// ---- FunctionBlocks/Sorter/Functions/FB_SorterLog.TcPOU
FUNCTION_BLOCK FB_SorterLog
VAR_IN_OUT
END_VAR
VAR_INPUT
	SorterToLog			:	ST_Sorter;
	SorterLogEnable		:	UDINT;
	ToInduct			:	ST_ItemTemporary;
END_VAR
VAR_OUTPUT
	TempItem			:	ST_ItemTemporary;
END_VAR
VAR
	rInductPE			:	R_TRIG;
	fInductPE			:	F_TRIG;
	rDischargePE		:	R_TRIG;
	fDischargePE		:	F_TRIG;
	sMessage			:	STRING;
	BlankItem			: 	ST_Item := (ID := ''
										, UniqueID := 0
										, Destination := 0
										, Status := E_StatusCode.No_Status
										, ExtStatus := E_StatusCode.No_Status
										, DeviceID := ''
										, MessageType := E_MessageIds.NoMessage_00);
END_VAR

// Capture rising and falling edge Triggers of the configured Sorter PE (Induct/Discharge)
rInductPE(CLK:= SorterToLog.InductPE, Q =>);
fInductPE(CLK:= SorterToLog.InductPE, Q =>);
rDischargePE(CLK:= SorterToLog.DischargePE, Q =>);
fDischargePE(CLK:= SorterToLog.DischargePE, Q =>);

// On the rising/falling edge of the Induct PE
IF rInductPE.Q OR fInductPE.Q THEN
	IF SorterLogEnable.SORTER_DISCHARGE_PE THEN
		// Write to the Error List
		ADSLOGSTR( msgCtrlMask := ADSLOG_MSGTYPE_HINT OR ADSLOG_MSGTYPE_LOG
			, msgFmtStr := CONCAT(sortertolog.Config.Name,' Induct PE Blocked : %s')
			, strArg := BOOL_TO_STRING(SorterToLog.InductPE)); 
	END_IF
END_IF

// Prepare a dummy record for items that arrive before BCR data is received
// On the rising edge of the Induct PE
IF rInductPE.Q THEN
	// Test for a UniqueID, which indicates that a Barcode has been received
	IF ToInduct.Item.UniqueID = 0 THEN
		// Capture and create relevant info
		TempItem.Counts := SorterToLog.EncoderCounts;
		TempItem.Item.UniqueID :=  UDINT_TO_DINT(SorterToLog.EncoderCounts);
		TempItem.Item.ID :=  CONCAT('T-', UDINT_TO_STRING(SorterToLog.EncoderCounts));
		TempItem.Item.Destination := SorterToLog.Config.DefaultDestination;
		TempItem.Item.DestinationIdx := SorterToLog.Config.DefaultDestIdx;
		TempItem.Item.Status := E_StatusCode.UnidentifiedItem;
		IF SorterLogEnable.SORTER_TEMPID THEN
			ADSLOGSTR( msgCtrlMask := ADSLOG_MSGTYPE_HINT OR ADSLOG_MSGTYPE_LOG
				, msgFmtStr := CONCAT(sortertolog.Config.Name,' Temp ID Assigned : %s')
				, strArg := TempItem.Item.ID);
		END_IF
	END_IF	
END_IF

// Clear the dummy record when the PE clears
// Items can only be inducted when the BCR info is received before or while the induct PE is blocked
IF fInductPE.Q THEN
	// Clear the record
	TempItem.Counts := 0;
	TempItem.Item :=  BlankItem;
END_IF

// On the rising/falling edge of the Discharge PE
IF rDischargePE.Q OR fDischargePE.Q THEN
	IF SorterLogEnable.SORTER_DISCHARGE_PE THEN
		// Write to the Error List
		ADSLOGSTR( msgCtrlMask := ADSLOG_MSGTYPE_HINT OR ADSLOG_MSGTYPE_LOG
			, msgFmtStr := CONCAT(sortertolog.Config.Name,' Discharge PE Blocked : %s')
			, strArg := BOOL_TO_STRING(SorterToLog.DischargePE)); 
	END_IF
END_IF

END_FUNCTION_BLOCK

// ---- FunctionBlocks/Divert/Functions/FB_DivertLog.TcPOU
FUNCTION_BLOCK FB_DivertLog
VAR_IN_OUT
	DivertArray	: ARRAY[*] OF ST_Divert;
END_VAR
VAR_INPUT
	DivertLogEnable		:	UDINT;
	EncoderCounts		:	UDINT;
END_VAR
VAR_OUTPUT
END_VAR
VAR
	DivertCountMax			: DINT;
	DivertCountMin			: DINT;
	DivertIndex				: DINT;
	r_DivertExtend			: ARRAY [1..16] OF R_TRIG;
	f_DivertExtend			: ARRAY [1..16] OF F_TRIG;
	r_ConfirmPE				: ARRAY [1..16] OF R_TRIG;
	f_ConfirmPE				: ARRAY [1..16] OF F_TRIG;
	sMessage				: STRING;
END_VAR

// Get the Max and Min counts
DivertCountMin := LOWER_BOUND(DivertArray,1);
DivertCountMax := UPPER_BOUND(DivertArray,1);

FOR DivertIndex := DivertCountMin TO DivertCountMax DO
	// Divert at DivertIndex
	r_DivertExtend[DivertIndex](CLK := DivertArray[DivertIndex].Output1);
	f_DivertExtend[DivertIndex](CLK := DivertArray[DivertIndex].Output1);
	
	IF r_DivertExtend[DivertIndex].Q THEN
		// Mask the divert index to see if it should be logged
		IF ((DivertLogEnable AND LREAL_TO_UDINT(EXPT(2,DivertIndex))) > 0) THEN
			sMessage := DINT_TO_STRING(DivertIndex);
			sMessage := CONCAT(sMessage,' : ');
			sMessage := CONCAT(sMessage, UDINT_TO_STRING(EncoderCounts));
			ADSLOGSTR( msgCtrlMask := ADSLOG_MSGTYPE_HINT OR ADSLOG_MSGTYPE_LOG
				, msgFmtStr := CONCAT(DivertArray[DivertIndex].Config.ID, ' Extend Divert %s')
				, strArg := sMessage); 
		END_IF;
	END_IF
	IF f_DivertExtend[DivertIndex].Q THEN
		// Mask the divert index to see if it should be logged
		IF ((DivertLogEnable AND LREAL_TO_UDINT(EXPT(2,DivertIndex))) > 0) THEN
			sMessage := DINT_TO_STRING(DivertIndex);
			sMessage := CONCAT(sMessage,' : ');
			sMessage := CONCAT(sMEssage, UDINT_TO_STRING(EncoderCounts));
			ADSLOGSTR( msgCtrlMask := ADSLOG_MSGTYPE_HINT OR ADSLOG_MSGTYPE_LOG
				, msgFmtStr := CONCAT(DivertArray[DivertIndex].Config.ID, ' Retract Divert %s')
				, strArg := sMessage); 
		END_IF;
	END_IF
	
	// Confirm at DivertIndex
	r_ConfirmPE[DivertIndex](CLK := DivertArray[DivertIndex].ConfirmPE);
	f_ConfirmPE[DivertIndex](CLK := DivertArray[DivertIndex].ConfirmPE);
	
	IF r_ConfirmPE[DivertIndex].Q THEN
		// Mask the convirm index to see if it should be logged
		IF ((DivertLogEnable AND LREAL_TO_UDINT(EXPT(2,(DivertIndex+15)))) > 0) THEN
			sMessage := DINT_TO_STRING(DivertIndex);
			sMessage := CONCAT(sMessage,' Blocked: ');
			sMessage := CONCAT(sMEssage, UDINT_TO_STRING(EncoderCounts));
			ADSLOGSTR( msgCtrlMask := ADSLOG_MSGTYPE_HINT OR ADSLOG_MSGTYPE_LOG
				, msgFmtStr := CONCAT(DivertArray[DivertIndex].Config.ID, ' Configm PE %s')
				, strArg := sMessage); 
		END_IF;
	END_IF
	IF f_ConfirmPE[DivertIndex].Q THEN
		// Mask the convirm index to see if it should be logged
		IF ((DivertLogEnable AND LREAL_TO_UDINT(EXPT(2,(DivertIndex+15)))) > 0) THEN
			sMessage := DINT_TO_STRING(DivertIndex);
			sMessage := CONCAT(sMessage,' Cleared: ');
			sMessage := CONCAT(sMEssage, UDINT_TO_STRING(EncoderCounts));
			ADSLOGSTR( msgCtrlMask := ADSLOG_MSGTYPE_HINT OR ADSLOG_MSGTYPE_LOG
				, msgFmtStr := CONCAT(DivertArray[DivertIndex].Config.ID, ' Configm PE %s')
				, strArg := sMessage); 
		END_IF;
	END_IF
END_FOR

END_FUNCTION_BLOCK

// ---- POUs/ProcessBuffers_P2140.TcPOU
PROGRAM ProcessBuffers_P2140
VAR_IN_OUT
	st_NextToInduct					: ST_ItemTemporary;
	st_UpdateItem					: ST_ItemTemporary;
	st_TempInductItem				: ST_ItemTemporary;
	{attribute 'OPC.UA.DA' := '0'}
	st_Sorter						: ST_Sorter;
	{attribute 'OPC.UA.DA' := '0'}
	aDiverts						: ARRAY[Sorter.DIVERTMIN_P2140..Sorter.NUMBEROFDIVERTS_P2140] OF ST_DIVERT;
	aItems 							: ARRAY[Sorter.SORTERENCODERMIN_P2140..Sorter.SORTERENCODERMAX_P2140] OF ST_Item;
END_VAR

VAR_INPUT
	DestinationOverride				: DINT;	// Pass in Divert to sent item to regardless of the direction received
	DivertToCommission				: DINT;
	ItemsArrayMax 					: UDINT;
	ItemsArrayMin 					: UDINT;
END_VAR

VAR_OUTPUT
	DefaultDestIdx					: DINT;
	RecircDestIdx					: DINT;
END_VAR

VAR
	fb_ArrivalBuffer				: FB_ItemBuffer;
	st_ArrivalItem 					: ST_Item;		// Arrival Item (Bar code read) from System PLC (BarCodeReaders.pou)

	// Item to replace in the sorter buffer
	st_ReplaceItem					: st_Item;

	fb_TransportBuffer				: FB_ItemBuffer;

	fb_UpdateBuffer 				: FB_ItemBuffer;

	st_ToUpdate						: ST_ItemTemporary;	// Item to Update on the Sorter, or waiting to be added to the sorter

	ItemsArraySize			: UDINT;

	TransportItemInSorter	: ST_Item;	// Temporary Processing Item
	TransportItemFound		: ST_Item;	// Item to Update Found
	TransportSorterIndex	: UDINT;

	ExitSorterIndex			: UDINT;
	ExitItemInSorter		: ST_Item;
	ExitItemFound			: ST_ItemTemporary;
	ExitInDivert			: BOOL;
	ExitDiverting			: BOOL;
	ExitSuccess				: BOOL;
	ExitDetected			: BOOL;
	ExitComplete			: BOOL;

	UpdateIndexCounter		: DINT;

	bTest : BOOL;
	sMessage	:	STRING;
	
	st_DisplayItem		:st_Item;
	LogSorterDump		:BOOL := FALSE;

	fb_FindDestination		: FB_FindDestination;
	fb_DefaultDestination	: FB_FindDestination;
	fb_RecircDestination	: FB_FindDestination;
	// Created to allow the aDiverts to be used in the FB_FindDestination Function Block
	{attribute 'OPC.UA.DA' := '0'}
	aTempDiverts			: ARRAY[Sorter.DIVERTMIN_P2140..Sorter.NUMBEROFDIVERTS_P2140] OF ST_DIVERT;
	
	nItemBufferLogEnable	:	UDINT;
	nSorterLogEnable		:	UDINT;
	nDivertLogEnable		:	UDINT;
	nSortBufferLogEnable	:	UDINT;
END_VAR

nItemBufferLogEnable := GVL_Logging.nItemBufferLogEnable OR GVL_Logging.nItemBufferLogEnableP2140;
nSorterLogEnable := GVL_Logging.nSorterLogEnable OR GVL_Logging.nSorterLogEnableP2140;
nDivertLogEnable := GVL_Logging.nDivertLogEnable OR GVL_Logging.nDivertLogEnableP2140;
nSortBufferLogEnable := GVL_Logging.nSortBufferLogEnable OR GVL_Logging.nSortBufferLogEnableP2140;

aTempDiverts := aDiverts;
// Initialize the Transport and Update buffers
// Set Master for FB's that control the buffer
fb_ArrivalBuffer.Master := FALSE;
fb_TransportBuffer.Master := FALSE;
fb_UpdateBuffer.Master := FALSE;

// Turn ON/OFF Logging of all activity in/out
fb_ArrivalBuffer.LogEntries := nItemBufferLogEnable.ARRIVALS;
fb_TransportBuffer.LogEntries := nItemBufferLogEnable.TRANSPORT;
fb_UpdateBuffer.LogEntries := nItemBufferLogEnable.UPDATE;

// Provide names for the buffers
fb_ArrivalBuffer.Name := CONCAT(st_Sorter.Config.Name, ' SRT ARRIVAL');
fb_TransportBuffer.Name := CONCAT(st_Sorter.Config.Name, ' SRT TRANSPORT');
fb_UpdateBuffer.Name := CONCAT(st_Sorter.Config.Name, ' SRT UPDATE');

// Initialize the FB_ItemExtBuffer Instances
fb_ArrivalBuffer(st_BufferData := st_SorterArrivalBuffer_P2140
						, st_BufferFdbkIn := st_ArrivalFdbkOut_P2140
						, st_BufferFdbkOut => st_ArrivalFdbkIn_P2140);
fb_TransportBuffer(st_BufferData := st_SorterTransportBuffer_P2140
						, st_BufferFdbkIn := st_TransportFdbkOut_P2140
						, st_BufferFdbkOut => st_TransportFdbkIn_P2140);
fb_UpdateBuffer(st_BufferData := st_SorterUpdateBuffer
						, st_BufferFdbkIn := st_UpdateFdbkOut
						, st_BufferFdbkOut => st_UpdateFdbkIn);

IF GVL_IO.INIT THEN
	fb_ArrivalBuffer.Clear();
	fb_TransportBuffer.Clear();
	fb_UpdateBuffer.Clear();
END_IF
						
(*
	Set the Upper/Lower bound of relevant arrays for looping purposes
	ItemsArrayMax/Min for the sorter array slot count
*)
// Size is Max - Min + 1 to capture both extremes
ItemsArraySize := ItemsArrayMax - ItemsArrayMin + 1;

(*
 	Check for a value disagreement in the Arrival Buffer In and Out pointers to
  	determine if there is an update for an item.
	When an Item arrives, the System PLC adds it to the shared buffer and increments
	the InPointer
*)
IF st_SorterArrivalBuffer_P2140.nInPointer <> fb_ArrivalBuffer.OutPointer THEN
	fb_ArrivalBuffer.RemoveItem(st_ItemToReturn => st_ArrivalItem);
END_IF

// Input Item read at bar code reader from System PLC to sorter
IF st_ArrivalItem.ID <> '' THEN
	IF nSortBufferLogEnable.BUFFER_ARRIVAL THEN
		sMessage := CONCAT('Item: ', st_ArrivalItem.ID);
		sMessage := CONCAT(sMessage,' Pulses: ');
		sMessage := CONCAT(sMessage, UDINT_TO_STRING(st_Sorter.EncoderCounts));
		// Write to the Error List
		ADSLOGSTR( msgCtrlMask := ADSLOG_MSGTYPE_HINT OR ADSLOG_MSGTYPE_LOG
			, msgFmtStr := CONCAT(st_Sorter.Config.Name, ' Arrival Processed: %s')
			, strArg := sMessage);
	END_IF
	// Indicate that this item did not get added to the sorter and add to the exit buffer
	//  Both as a TransportUpdate and TransportComplete message type 
	IF st_NextToInduct.Item.ID <> '' THEN
		IF nSortBufferLogEnable.BUFFER_MISSINDUCT THEN
			sMessage := CONCAT('Item: ', st_NextToInduct.Item.ID);
			// Write to the Error List
			ADSLOGSTR( msgCtrlMask := ADSLOG_MSGTYPE_HINT OR ADSLOG_MSGTYPE_LOG
				, msgFmtStr := CONCAT(st_Sorter.Config.Name, ' Item Removed - Not Inducted: %s')
				, strArg := sMessage);
		END_IF
		// Transport Response
		st_NextToInduct.Item.Status := E_StatusCode.Assign_NotInducted;
		st_NextToInduct.Item.DeviceID := st_Sorter.Config.EquipID;
		st_NextToInduct.Item.MessageType := E_MessageIds.TransportResponse_25;
		fb_UpdateBuffer.AddItem(st_ItemToAdd := st_NextToInduct.Item);

		// Transport Complete
		st_NextToInduct.Item.Status := E_StatusCode.Divert_NotInducted;
		st_NextToInduct.Item.MessageType := E_MessageIds.TransportComplete_26;
		fb_UpdateBuffer.AddItem(st_ItemToAdd := st_NextToInduct.Item);
	END_IF
	// Copy Last BCR item to Item to Induct
	st_NextToInduct.Item :=  st_ArrivalItem;
	// Add the Sorter EquipID to the NextToInduct
	st_NextToInduct.Item.DeviceID := st_Sorter.Config.EquipID;
	// Set the Default Destination
	IF DestinationOverride = 0 THEN
		st_NextToInduct.Item.Destination := st_Sorter.Config.DefaultDestination;
		st_NextToInduct.Item.DestinationIdx := st_Sorter.Config.DefaultDestIdx;
	ELSE
		st_NextToInduct.Item.Destination := DestinationOverride;
		IF nSorterLogEnable.SORTER_DESTINATION_LU THEN
			sMessage := CONCAT('Destination: ', DINT_TO_STRING(st_NextToInduct.Item.Destination));
			// Write to the Error List
			ADSLOGSTR( msgCtrlMask := ADSLOG_MSGTYPE_HINT OR ADSLOG_MSGTYPE_LOG
				, msgFmtStr := CONCAT(st_sorter.Config.Name, ' Buffer Destination OR Lookup %s')
				, strArg := sMessage);
		END_IF
		fb_FindDestination(RoundRobin := st_Sorter.RoundRobin
						, SorterLogEnable := nSorterLogEnable
						, aDiverts := aTempDiverts
						, DestinationID := st_NextToInduct.Item.Destination
						, DestinationIndex => st_NextToInduct.Item.DestinationIdx);
		
	END_IF
	// Capture an encoder value that when the encoder count exceeds this value, NextToInduct item will be cleared
	st_NextToInduct.Counts := st_Sorter.EncoderCounts;
	// Clear the Last recieved item
	st_ArrivalItem := BlankItem;
	// Prepare to replace the Temporarily assigned item with this item
	IF st_TempInductItem.Item.ID <> '' THEN
		// Capture the Counts and Length from the temporary item
		st_NextToInduct.Counts := st_TempInductItem.Counts;
		st_NextToInduct.Item.Length := st_TempInductItem.Item.Length;
		//Identify the Item to replace in the sorter array
		st_ReplaceItem := st_TempInductItem.Item;
		st_TempInductItem.Counts := 0;
		st_TempInductItem.Item := BlankItem;
		IF nSortBufferLogEnable.BUFFER_TEMPINDUCT THEN
			ADSLOGSTR( msgCtrlMask := ADSLOG_MSGTYPE_HINT OR ADSLOG_MSGTYPE_LOG
				, msgFmtStr := CONCAT(st_Sorter.Config.Name, ' Temp ID Replaced : %s')
				, strArg := st_ReplaceItem.ID); 
		END_IF
	END_IF
END_IF

(*
 	Check for a value disagreement in the SorterTransportBuffer In and Out pointers to
  	determine if there is an update for an item.
	When an update arrived, the System PLC adds it to the shared buffer and increments
	the InPointer
*)
IF st_SorterTransportBuffer_P2140.nInPointer <> fb_TransportBuffer.OutPointer THEN
	fb_TransportBuffer.RemoveItem(st_ItemToReturn => st_ToUpdate.Item);
	// Override any received destination if there is an Override
	IF DestinationOverride <> 0 THEN
		st_ToUpdate.Item.Destination := DestinationOverride;
	END_IF
	// Lookup the index for the chosen destination
	IF nSorterLogEnable.SORTER_DESTINATION_LU THEN
		sMessage := CONCAT('Destination: ', DINT_TO_STRING(st_ToUpdate.Item.Destination));
		// Write to the Error List
		ADSLOGSTR( msgCtrlMask := ADSLOG_MSGTYPE_HINT OR ADSLOG_MSGTYPE_LOG
			, msgFmtStr := CONCAT(st_sorter.Config.Name, ' Buffer Update Lookup %s')
			, strArg := sMessage);
	END_IF
	fb_FindDestination(RoundRobin := st_Sorter.RoundRobin
					, SorterLogEnable := nSorterLogEnable
					, aDiverts := aTempDiverts
					, DestinationID := st_ToUpdate.Item.Destination
					, DestinationIndex => st_ToUpdate.Item.DestinationIdx);
	IF nSortBufferLogEnable.BUFFER_DESTINDEX THEN
		sMessage := CONCAT('Item: ', st_ToUpdate.Item.ID);
		sMessage := CONCAT(sMessage,' Destination: ');
		sMessage := CONCAT(sMessage, DINT_TO_STRING(st_ToUpdate.Item.Destination));
		sMessage := CONCAT(sMessage,' Index: ');
		sMessage := CONCAT(sMessage, DINT_TO_STRING(st_ToUpdate.Item.DestinationIdx));
		// Write to the Error List
		ADSLOGSTR( msgCtrlMask := ADSLOG_MSGTYPE_HINT OR ADSLOG_MSGTYPE_LOG
			, msgFmtStr := CONCAT(st_Sorter.Config.Name, ' Divert Index of Destination: %s')
			, strArg := sMessage);
	END_IF
END_IF

// Get the Default Destination Index
fb_DefaultDestination(RoundRobin := st_Sorter.RoundRobin
				, NoAssignment := TRUE
				, aDiverts := aTempDiverts
				, DestinationID := st_Sorter.Config.DefaultDestination
				, DestinationIndex => DefaultDestIdx);

// Get the Recirculation Destination Index
fb_RecircDestination(RoundRobin := st_Sorter.RoundRobin
				, NoAssignment := TRUE
				, aDiverts := aTempDiverts
				, DestinationID := st_Sorter.Config.RecircDestination
				, DestinationIndex => RecircDestIdx);

// Test the Item to Update against the Item to Induct and update if they match:
//	Update the NextItemToInduct with the updated data, then clear the Item to Update
IF st_ToUpdate.Item.ID <> '' THEN
	IF st_ToUpdate.Item.ID = st_NextToInduct.Item.ID THEN
		// Indicate that the transport command was received and a response was sent
		st_NextToInduct.Item.MessageType := E_MessageIds.TransportResponse_25;
		// Test the assigned lane for availability
		IF (aDiverts[st_ToUpdate.Item.DestinationIdx].Full
		   OR aDiverts[st_ToUpdate.Item.DestinationIdx].Faulted)
		   AND DestinationOverride = 0
		   THEN
			// Prepare a message to indicate that the item cannot be assigned
			st_ToUpdate.Item.Status := E_StatusCode.Assign_Full;
			st_ToUpdate.Item.DeviceID := st_Sorter.Config.EquipID;
			st_ToUpdate.Item.MessageType := E_MessageIds.TransportResponse_25;
			fb_UpdateBuffer.AddItem(st_ItemToAdd := st_ToUpdate.Item);
			st_NextToInduct.Item.ExtStatus := E_StatusCode.Divert_Full;
		ELSE
			st_NextToInduct.Item.DeviceID := st_Sorter.Config.EquipID;
			st_NextToInduct.Item.Status := E_StatusCode.Assign_Accepted;
			// Update the Destination
			st_NextToInduct.Item.Destination := st_ToUpdate.Item.Destination;
			st_NextToInduct.Item.DestinationIdx := st_ToUpdate.Item.DestinationIdx;
			fb_UpdateBuffer.AddItem(st_ItemToAdd := st_NextToInduct.Item);
		END_IF
		// If commissioning, ignore any other direction
		IF DivertToCommission > 0 THEN
			st_NextToInduct.Item.Destination := DivertToCommission;
		END_IF
		// Log the update
		IF nSortBufferLogEnable.BUFFER_INDUCT THEN
			sMessage := CONCAT('Item: ', st_ToUpdate.Item.ID);
			sMessage := CONCAT(sMessage,' Pulses: ');
			sMessage := CONCAT(sMessage, UDINT_TO_STRING(st_Sorter.EncoderCounts));
			sMessage := CONCAT(sMessage,' Status: ');
			sMessage := CONCAT(sMessage, UDINT_TO_STRING(st_ToUpdate.Item.Status));
			sMessage := CONCAT(sMessage,' Ext Status: ');
			sMessage := CONCAT(sMessage, UDINT_TO_STRING(st_ToUpdate.Item.ExtStatus));
			// Write to the Error List
			ADSLOGSTR( msgCtrlMask := ADSLOG_MSGTYPE_HINT OR ADSLOG_MSGTYPE_LOG
				, msgFmtStr := CONCAT(st_Sorter.Config.Name, ' Found Before Induct: %s')
				, strArg := sMessage);
		END_IF
		// We updated the item we were inducting, clear the Item to update
		st_ToUpdate.Item := BlankItem;
	END_IF
END_IF

// Clear the Update Item Found record each pass
TransportItemFound := BlankItem;

// Clear the last detected Exit item
ExitItemFound.Item := BlankItem;

// Reset the Detection booleans
ExitInDivert := FALSE;
ExitDiverting := FALSE;
ExitDetected := FALSE;
ExitSuccess := FALSE;
ExitComplete := FALSE;

// Loop through the entire array, it should be appropriately sized for the length of the sorter section
FOR UpdateIndexCounter := UDINT_TO_DINT(ItemsArrayMin) TO UDINT_TO_DINT(ItemsArrayMax) DO //Loop through everything in the sorter	

	// For Transport commands, start from the current encoder count and work forwards, just like the exit
	TransportSorterIndex := F_CalculateIndex(Offset := (UpdateIndexCounter)
											, InitialValue := st_Sorter.EncoderCounts
											, BufferSize := ItemsArraySize);

	// This is the item in the sorter array that we will be procesing this pass, testing for a Transport update message
	TransportItemInSorter := aItems[UDINT_TO_DINT(TransportSorterIndex)];

	// Test for a replace item
	// ReplaceItem is the temporary item
	// NextToInduct is the item to replace the temporary with
	IF st_ReplaceItem.ID <> '' THEN
		IF st_ReplaceItem.ID = TransportItemInSorter.ID THEN
			IF nSortBufferLogEnable.BUFFER_REPLACEINDUCT THEN
				sMessage := CONCAT('Item: ', st_ReplaceItem.ID);
				sMessage := CONCAT(sMessage,' New Item: ');
				sMessage := CONCAT(sMessage, st_NextToInduct.Item.ID);
				sMessage := CONCAT(sMessage,' Index: ');
				sMessage := CONCAT(sMessage, UDINT_TO_STRING(TransportSorterIndex));
				sMessage := CONCAT(sMessage,' Orig Dest: ');
				sMessage := CONCAT(sMessage, DINT_TO_STRING(TransportItemInSorter.Destination));
				sMessage := CONCAT(sMessage,' New Dest: ');
				sMessage := CONCAT(sMEssage, DINT_TO_STRING(st_ReplaceItem.Destination));
				sMessage := CONCAT(sMessage,' Orig Idx: ');
				sMessage := CONCAT(sMessage, DINT_TO_STRING(TransportItemInSorter.DestinationIdx));
				sMessage := CONCAT(sMessage,' New Idx: ');
				sMessage := CONCAT(sMEssage, DINT_TO_STRING(st_ReplaceItem.DestinationIdx));
				// Write to the Error List
				ADSLOGSTR( msgCtrlMask := ADSLOG_MSGTYPE_HINT OR ADSLOG_MSGTYPE_LOG
					, msgFmtStr := CONCAT(st_Sorter.Config.Name, ' Item ID Replaced After Induct: %s')
					, strArg := sMessage);
			END_IF
			TransportItemInSorter.ID := st_NextToInduct.Item.ID;
			TransportItemInSorter.Destination := st_NextToInduct.Item.Destination;
			TransportItemInSorter.DestinationIdx := st_NextToInduct.Item.DestinationIdx;
			TransportItemInSorter.DeviceID := st_NextToInduct.Item.DeviceID;
			TransportItemInSorter.MessageType := st_NextToInduct.Item.MessageType;
			TransportItemInSorter.Status := st_NextToInduct.Item.Status;
			TransportItemInSorter.UniqueID := st_NextToInduct.Item.UniqueID;
			TransportItemInSorter.CapturedInMetrics := st_NextToInduct.Item.CapturedInMetrics;
		END_IF
	END_IF
	// Test for an Item Update
	IF st_ToUpdate.Item.ID <> '' THEN
		// Test the sorter item against the update item
		IF st_ToUpdate.Item.ID = TransportItemInSorter.ID THEN
			IF nSortBufferLogEnable.BUFFER_UPDATEINDUCT THEN
				sMessage := CONCAT('Item: ', st_ToUpdate.Item.ID);
				sMessage := CONCAT(sMessage,' Index: ');
				sMessage := CONCAT(sMessage, UDINT_TO_STRING(TransportSorterIndex));
				// Write to the Error List
				ADSLOGSTR( msgCtrlMask := ADSLOG_MSGTYPE_HINT OR ADSLOG_MSGTYPE_LOG
					, msgFmtStr := CONCAT(st_Sorter.Config.Name, ' Found After Induct: %s')
					, strArg := sMessage);
			END_IF
			// Copy the found item record, 
			TransportItemFound := TransportItemInSorter;
			// Test the destined divert for availability
			IF aDiverts[st_ToUpdate.Item.DestinationIdx].Full OR aDiverts[st_ToUpdate.Item.DestinationIdx].Faulted THEN
				// Prepare a message to indicate that the item cannot be assigned
				TransportItemFound.Status := E_StatusCode.Assign_Full;
				TransportItemFound.ExtStatus := E_StatusCode.Divert_Full;
				TransportItemFound.MessageType := E_MessageIds.TransportResponse_25;
				TransportItemFound.Destination := st_Sorter.Config.DefaultDestination;
				TransportItemFound.DestinationIdx := st_Sorter.Config.DefaultDestIdx;
			// Test for an already diverting item and assign an ExtStatus of LateAssignment
			ELSIF TransportItemInSorter.Status >= E_StatusCode.Diverting THEN
				TransportItemFound.ExtStatus := E_StatusCode.Divert_LateAssignment;
				TransportItemFound.MessageType := E_MessageIds.TransportResponse_25;
			ELSE
				//  Change the destination, which should be the only item in the update
				TransportItemFound.Destination := st_ToUpdate.Item.Destination;
				TransportItemFound.DestinationIdx := st_ToUpdate.Item.DestinationIdx;
				// This message indicates we could assign the Item
				TransportItemFound.Status := E_StatusCode.Assign_Accepted;
				TransportItemFound.MessageType := E_MessageIds.TransportResponse_25;
			END_IF
			TransportItemFound.DeviceID := st_Sorter.Config.EquipID;
			// Add the item to the update buffer
			fb_UpdateBuffer.AddItem(TransportItemFound);
			// Clear the ToUpdate Item
			st_ToUpdate.Item := BlankItem;
		END_IF
	END_IF
	
	IF TransportItemFound.ID <> '' THEN
		// Test the sorter item against the update item
		IF TransportItemFound.ID = TransportItemInSorter.ID THEN
			// Only update if it is different
			IF TransportItemFound.Destination <> TransportItemInSorter.Destination THEN
				IF nSortBufferLogEnable.BUFFER_UPDATEDEST THEN
					sMessage := CONCAT('Item: ', TransportItemInSorter.ID);
					sMessage := CONCAT(sMessage,' Index: ');
					sMessage := CONCAT(sMessage, UDINT_TO_STRING(TransportSorterIndex));
					sMessage := CONCAT(sMessage,' Orig Dest: ');
					sMessage := CONCAT(sMessage, DINT_TO_STRING(TransportItemInSorter.Destination));
					sMessage := CONCAT(sMessage,' Orig Idx: ');
					sMessage := CONCAT(sMessage, DINT_TO_STRING(TransportItemInSorter.DestinationIdx));
					sMessage := CONCAT(sMessage,' Orig DeviceID ');
					sMessage := CONCAT(sMessage, TransportItemInSorter.DeviceID);
					// Write to the Error List
					ADSLOGSTR( msgCtrlMask := ADSLOG_MSGTYPE_HINT OR ADSLOG_MSGTYPE_LOG
						, msgFmtStr := CONCAT(st_Sorter.Config.Name, ' Dest Updated After Induct: %s')
						, strArg := sMessage);
				END_IF
				// Update the Destination. If the destination is unavailable, it has been already been set to the default
				TransportItemInSorter.Destination := TransportItemFound.Destination;
				TransportItemInSorter.DestinationIdx := TransportItemFound.DestinationIdx;
				TransportItemInSorter.DeviceID := TransportItemFound.DeviceID;
				TransportItemInSorter.MessageType := TransportItemFound.MessageType;
				TransportItemInSorter.Status := TransportItemFound.Status;
				TransportItemInSorter.ExtStatus := TransportItemFound.ExtStatus;
	
				IF nSortBufferLogEnable.BUFFER_UPDATEDEST THEN
					sMessage := CONCAT('Item: ', TransportItemInSorter.ID);
					sMessage := CONCAT(sMessage,' Index: ');
					sMessage := CONCAT(sMessage, UDINT_TO_STRING(TransportSorterIndex));
					sMessage := CONCAT(sMessage,' New Dest: ');
					sMessage := CONCAT(sMessage, DINT_TO_STRING(TransportItemInSorter.Destination));
					sMessage := CONCAT(sMessage,' New Idx: ');
					sMessage := CONCAT(sMessage, DINT_TO_STRING(TransportItemInSorter.DestinationIdx));
					sMessage := CONCAT(sMessage,' New DeviceID ');
					sMessage := CONCAT(sMessage, TransportItemInSorter.DeviceID);
					// Write to the Error List
					ADSLOGSTR( msgCtrlMask := ADSLOG_MSGTYPE_HINT OR ADSLOG_MSGTYPE_LOG
						, msgFmtStr := CONCAT(st_Sorter.Config.Name, ' Dest Updated After Induct: %s')
						, strArg := sMessage);
				END_IF
			END_IF
			// Make sure that the destination update makes it to the item being inducted into the sorter
			IF st_UpdateItem.Item.ID <> '' THEN
				IF st_UpdateItem.Item.ID = TransportItemFound.ID THEN
					IF st_UpdateItem.Item.Destination <> TransportItemFound.Destination THEN
						IF nSortBufferLogEnable.BUFFER_UPDATEDEST THEN
							// Log the original destination
							sMessage := CONCAT('Item: ', st_UpdateItem.Item.ID);
							sMessage := CONCAT(sMessage, ' Pulses: ');
							sMessage := CONCAT(sMessage, UDINT_TO_STRING(st_Sorter.EncoderCounts));
							sMessage := CONCAT(sMessage,' Orig Dest: ');
							sMessage := CONCAT(sMessage, DINT_TO_STRING(st_UpdateItem.Item.Destination));
							sMessage := CONCAT(sMessage,' Orig Idx: ');
							sMessage := CONCAT(sMessage, DINT_TO_STRING(st_UpdateItem.Item.DestinationIdx));
							// Write to the Error List
							ADSLOGSTR( msgCtrlMask := ADSLOG_MSGTYPE_HINT OR ADSLOG_MSGTYPE_LOG
								, msgFmtStr := CONCAT(st_Sorter.Config.Name, ' Induct Dest Changed: %s')
								, strArg := sMessage);
						END_IF
						// Update the Destination and Index
						st_UpdateItem.Item.Destination := TransportItemFound.Destination;
						st_UpdateItem.Item.DestinationIdx := TransportItemFound.DestinationIdx;
						// Log the new destination
						IF nSortBufferLogEnable.BUFFER_UPDATEDEST THEN
							sMessage := CONCAT('Item: ', st_UpdateItem.Item.ID);
							sMessage := CONCAT(sMessage, ' Pulses: ');
							sMessage := CONCAT(sMessage, UDINT_TO_STRING(st_Sorter.EncoderCounts));
							sMessage := CONCAT(sMessage,' New Dest: ');
							sMessage := CONCAT(sMessage, DINT_TO_STRING(st_UpdateItem.Item.Destination));
							sMessage := CONCAT(sMessage,' New Idx: ');
							sMessage := CONCAT(sMessage, DINT_TO_STRING(st_UpdateItem.Item.DestinationIdx));
							// Write to the Error List
							ADSLOGSTR( msgCtrlMask := ADSLOG_MSGTYPE_HINT OR ADSLOG_MSGTYPE_LOG
								, msgFmtStr := CONCAT(st_Sorter.Config.Name, ' Induct Dest Changed: %s')
								, strArg := sMessage);
						END_IF
					END_IF
				END_IF
			ELSE
				IF nSortBufferLogEnable.BUFFER_UPDATEDEST THEN
					sMessage := CONCAT('Item: ', TransportItemInSorter.ID);
					sMessage := CONCAT(sMessage,' Index: ');
					sMessage := CONCAT(sMessage, UDINT_TO_STRING(TransportSorterIndex));
					sMessage := CONCAT(sMessage,' Orig Dest: ');
					sMessage := CONCAT(sMessage, DINT_TO_STRING(TransportItemInSorter.Destination));
					sMessage := CONCAT(sMessage,' Orig Idx: ');
					sMessage := CONCAT(sMessage, DINT_TO_STRING(TransportItemInSorter.DestinationIdx));
					// Write to the Error List
					ADSLOGSTR( msgCtrlMask := ADSLOG_MSGTYPE_HINT OR ADSLOG_MSGTYPE_LOG
						, msgFmtStr := CONCAT(st_Sorter.Config.Name, ' Dest Received After Induct: %s')
						, strArg := sMessage);
				END_IF
			END_IF
		END_IF
	END_IF

	// Put the updated record back into the array
	aItems[TransportSorterIndex] := TransportItemInSorter;
	
//==================================================
// 	Done procesing Transport information
//
//	Begin processing Update/Exit information
//==================================================
	
	// For exits, start from the current encoder count and work forward
	ExitSorterIndex := F_CalculateIndex(Offset := UpdateIndexCounter
										, InitialValue := st_Sorter.EncoderCounts
										, BufferSize := ItemsArraySize);

	// Identify the Item we are testing
	ExitItemInSorter := aItems[ExitSorterIndex];

	// Populated ID identifies an item in the sorter
	// Between the two Divert status codes indicates that the item has attempted to divert
	IF ExitItemInSorter.ID <> '' THEN
		// Capture the Item encoder index and the Item at the current index
		//  This represents the first item record for this item
		//  It is captured to log the start index to allow this first record to be updated
		//  when the item is completely diverted
		IF ExitItemFound.Item.ID = '' THEN
			ExitItemFound.Counts := ExitSorterIndex;
			ExitItemFound.Item := ExitItemInSorter;
			IF ExitItemFound.Item.Status = E_StatusCode.Divert_Complete THEN
				ExitComplete := TRUE;
			END_IF
		END_IF
		// When ExitComplete is TRUE, and the ID's match, clear out this Item
		IF ExitComplete THEN
			IF ExitItemInSorter.ID = ExitItemFound.Item.ID THEN
				IF aItems[ExitSorterIndex].ID <> '' THEN
					IF nSortBufferLogEnable.BUFFER_DUMP THEN
						sMessage := CONCAT('Item: ', aItems[ExitSorterIndex].ID);
						sMessage := CONCAT(sMessage,' Index: ');
						sMessage := CONCAT(sMessage, UDINT_TO_STRING(ExitSorterIndex));
						sMessage := CONCAT(sMessage,' Item Status: ');
						sMessage := CONCAT(sMessage, DINT_TO_STRING(aItems[ExitSorterIndex].Status));
						sMessage := CONCAT(sMessage,' Item Ext Status: ');
						sMessage := CONCAT(sMessage, DINT_TO_STRING(aItems[ExitSorterIndex].ExtStatus));
						// Write to the Error List
						ADSLOGSTR( msgCtrlMask := ADSLOG_MSGTYPE_HINT OR ADSLOG_MSGTYPE_LOG
							, msgFmtStr := CONCAT(st_Sorter.Config.Name, ' Exit Complete Dump Info: %s')
							, strArg := sMessage);
					END_IF
				END_IF
				aItems[ExitSorterIndex] := BlankItem;
			END_IF
		// When ExitComplete is FALSE, test for a diverting/diverted item
		ELSE
			// Detect when this item is in a diverting state
			IF (ExitItemInSorter.Status >= E_StatusCode.Diverting
			   OR ExitItemInSorter.Status <= E_StatusCode.Divert_Success)
			   THEN
			   	ExitInDivert := TRUE;
				(*
					Status value increase from Diverting to Divert_Complete
					Codes to indicate divert disposition are between Diverting and Divert_Detected
					Divert_Full and Diverting are set in FB_DivertDecision/FB_DivertControl
					Divert_Detected, Divert_Success, and Divert_Missed are set in FB_ConfirmCheck
				*)
				ExitDiverting := TRUE;
				IF ExitItemInSorter.Status = E_StatusCode.Divert_Detected THEN
					ExitDetected := TRUE;
				END_IF
				// Once the divert is successful, we are no longer "diverting"
				IF ExitItemInSorter.Status = E_StatusCode.Divert_Success THEN
					ExitSuccess := TRUE;
					ExitDiverting := FALSE;
				END_IF
				(*	
					ExitItemInSorter is the current item being examined
					ExitItemFound.Item is a copy of the Array item at ExitItemFound.Counts
					ExitItemFound.Counts references the Array index of the first record associated with this item
					When a Status/ExtStatus of greater value is detected, the first record Status/ExtStatus is overwritten
					The ExitItemFound.Item.Status/.ExtStatus is also updated
				*)
				IF ExitItemInSorter.Status > aItems[ExitItemFound.Counts].Status THEN
					aItems[ExitItemFound.Counts].Status := ExitItemInSorter.Status;
					ExitItemFound.Item.Status := ExitItemInSorter.Status;
				END_IF
				IF ExitItemInSorter.ExtStatus > aItems[ExitItemFound.Counts].ExtStatus THEN
					aItems[ExitItemFound.Counts].ExtStatus := ExitItemInSorter.ExtStatus;
					ExitItemFound.Item.ExtStatus := ExitItemInSorter.ExtStatus;
				END_IF
			END_IF
			aItems[ExitSorterIndex].Status := ExitItemFound.Item.Status;
		END_IF
	ELSE
		(*
			This path is followed when the ExitItemInSorter.ID is empty, which indicates
			that the array record associated with this index is not occupied

			ExitInDivert, ExitDiverting and ExitSuccess are all set while the .ID is not empty
		*)
		// This item was in a "diverting" state
		IF ExitInDivert THEN
			// This item is not currently diverting
			IF NOT ExitDiverting THEN
				// Only change to a Divert_Success if a Divert_Success was detected
				// Any other status is captured in the ELSE clause of the CASE statement
				IF ExitSuccess THEN
					ExitItemFound.Item.Status := E_StatusCode.Divert_Success;
				END_IF
				IF NOT (ExitItemFound.Item.DestinationIdx = Sorter.NUMBEROFDIVERTS_P2140)
				   OR (ExitItemFound.Item.DestinationIdx = Sorter.NUMBEROFDIVERTS_P2140 AND aDiverts[ExitItemFound.Item.DestinationIdx].Config.IsDischarge)
				   THEN 
					ExitItemFound.Item.CapturedInMetrics := TRUE;
					ExitItemFound.Item.MessageType := E_MessageIds.TransportComplete_26;
					fb_UpdateBuffer.AddItem(ExitItemFound.Item);
					aItems[ExitItemFound.Counts].Status := E_StatusCode.Divert_Complete;
				END_IF
			END_IF
		END_IF
		// Clear the last detected Exit item
		ExitItemFound.Item := BlankItem;
		// Reset the Detection booleans
		ExitInDivert := FALSE;
		ExitDiverting := FALSE;
		ExitDetected := FALSE;
		ExitSuccess := FALSE;
		ExitComplete := FALSE;
	END_IF
END_FOR

// If the ID is populated, we didn't find a match to update
IF st_ToUpdate.Item.ID <> '' THEN
	IF nSortBufferLogEnable.BUFFER_UNASSIGNED THEN
		sMessage := CONCAT('Item: ', st_ToUpdate.Item.ID);
		// Write to the Error List
		ADSLOGSTR( msgCtrlMask := ADSLOG_MSGTYPE_HINT OR ADSLOG_MSGTYPE_LOG
			, msgFmtStr := CONCAT(st_Sorter.Config.Name, ' Item Not Updated: %s')
			, strArg := sMessage);
	END_IF
	st_ToUpdate.Item.Status := E_StatusCode.Assign_NotFound;
	st_ToUpdate.Item.DeviceID := st_Sorter.Config.Name;
	st_ToUpdate.Item.MessageType := E_MessageIds.TransportResponse_25;
	fb_UpDateBuffer.AddItem(st_ItemToAdd := st_ToUpdate.Item);
	st_ToUpdate.Item := BlankItem;
END_IF

END_PROGRAM

// ---- FunctionBlocks/Sorter/Functions/FB_FindDestination.TcPOU
FUNCTION_BLOCK FB_FindDestination
VAR_IN_OUT
	RoundRobin		:	ST_RoundRobin;
	aDiverts		:	ARRAY[*] OF ST_Divert;
	DestinationID	:	DINT;
END_VAR
VAR_INPUT
	SorterLogEnable	:	UDINT;
	NoAssignment		:	BOOL;
END_VAR
VAR_OUTPUT
	DestinationIndex	:	DINT;
	DestinationState	:	DINT;
END_VAR
VAR
	DivertArrayMin		:	DINT;
	DivertArrayMax		:	DINT;
	Last_Enabled		:	UINT;
	IndexCheck			:	DINT;
	sMessage			:	STRING;
	CheckEnableAvail	:	DINT;
	Enabled				:	UINT;
	Available			:	UINT;
END_VAR

// Get the upper and lower bounds of the divert array
DivertArrayMin := LOWER_BOUND(aDiverts,1);
DivertArrayMax := UPPER_BOUND(aDiverts,1);

//When a response is received, find the designated Destination
IF DestinationID >= 0 THEN
	IF SorterLogEnable.SORTER_DESTINATION_LU THEN
		sMessage := CONCAT('Destination: ', DINT_TO_STRING(DestinationID));
		// Write to the Error List
		ADSLOGSTR( msgCtrlMask := ADSLOG_MSGTYPE_HINT OR ADSLOG_MSGTYPE_LOG
			, msgFmtStr := 'Lookup %s'
			, strArg := sMessage);
	END_IF
	// Check to see if the Destination is defined as a round-robin destination for this sorter
	IF DestinationID = RoundRobin.Config.Destination THEN
		// Set Enabled
		Enabled.0 := RoundRobin.Config.Destinations[0].Enabled;
		Enabled.1 := RoundRobin.Config.Destinations[1].Enabled;
		Enabled.2 := RoundRobin.Config.Destinations[2].Enabled;
		Enabled.3 := RoundRobin.Config.Destinations[3].Enabled;
		Enabled.4 := RoundRobin.Config.Destinations[4].Enabled;
		Enabled.5 := RoundRobin.Config.Destinations[5].Enabled;
		Enabled.6 := RoundRobin.Config.Destinations[6].Enabled;
		Enabled.7 := RoundRobin.Config.Destinations[7].Enabled;
		Enabled.8 := RoundRobin.Config.Destinations[8].Enabled;
		Enabled.9 := RoundRobin.Config.Destinations[9].Enabled;
		Enabled.10 := RoundRobin.Config.Destinations[10].Enabled;
		Enabled.11 := RoundRobin.Config.Destinations[11].Enabled;
		Enabled.12 := RoundRobin.Config.Destinations[12].Enabled;
		Enabled.13 := RoundRobin.Config.Destinations[13].Enabled;
		Enabled.14 := RoundRobin.Config.Destinations[14].Enabled;
		Enabled.15 := RoundRobin.Config.Destinations[15].Enabled;
		// Set Available
		Available.0 := RoundRobin.Config.Destinations[0].Available;
		Available.1 := RoundRobin.Config.Destinations[1].Available;
		Available.2 := RoundRobin.Config.Destinations[2].Available;
		Available.3 := RoundRobin.Config.Destinations[3].Available;
		Available.4 := RoundRobin.Config.Destinations[4].Available;
		Available.5 := RoundRobin.Config.Destinations[5].Available;
		Available.6 := RoundRobin.Config.Destinations[6].Available;
		Available.7 := RoundRobin.Config.Destinations[7].Available;
		Available.8 := RoundRobin.Config.Destinations[8].Available;
		Available.9 := RoundRobin.Config.Destinations[9].Available;
		Available.10 := RoundRobin.Config.Destinations[10].Available;
		Available.11 := RoundRobin.Config.Destinations[11].Available;
		Available.12 := RoundRobin.Config.Destinations[12].Available;
		Available.13 := RoundRobin.Config.Destinations[13].Available;
		Available.14 := RoundRobin.Config.Destinations[14].Available;
		Available.15 := RoundRobin.Config.Destinations[15].Available;
		// Test to see if the last enabled round robin destinations are still enabled
		// If they are different, restart the round-robin assignment to accommodate differences 
		IF Enabled = Last_Enabled THEN
			// Test to see if the round robin assignments have all been met
			// If they have, clear and start over
			IF Available = RoundRobin.Sent THEN
				RoundRobin.Sent := 0;
			END_IF
		ELSE
			// Capture the new enabled round-robin destinations
			// Restart the round robin assignments
			Last_Enabled := Enabled;
			RoundRobin.Sent := 0;
		END_IF
		FOR IndexCheck := 0 TO 15 DO
			IF (
			   ((Enabled AND LREAL_TO_UINT(EXPT(2,IndexCheck))) > 0) 
			   AND ((Available AND LREAL_TO_UINT(EXPT(2,IndexCheck))) > 0)
			   AND NOT ((RoundRobin.Sent AND LREAL_TO_UINT(EXPT(2,IndexCheck))) > 0))
			   THEN
				IF NOT NoAssignment THEN
					RoundRobin.Sent := LREAL_TO_UINT(EXPT(2,IndexCheck)) OR RoundRobin.Sent;
					DestinationID := RoundRobin.Config.Destinations[IndexCheck].aDestination;
					IF SorterLogEnable.SORTER_DESTINATION_LU THEN
						sMessage := DINT_TO_STRING(DestinationIndex);
						sMessage := CONCAT('Dest ID: ', DINT_TO_STRING(DestinationID));
						// Write to the Error List
						ADSLOGSTR( msgCtrlMask := ADSLOG_MSGTYPE_HINT OR ADSLOG_MSGTYPE_LOG
							, msgFmtStr := 'RoundRobin %s'
							, strArg := sMessage);
					END_IF
				END_IF
				DestinationState := 0;
				EXIT;
			END_IF
		END_FOR
	END_IF
	// Always find the index for the destination, whether Round robin or assigned
	DestinationIndex := DivertArrayMax;
	FOR IndexCheck := DivertArrayMin TO DivertArrayMax  DO
		IF aDiverts[IndexCheck].Config.Number = DestinationID THEN
			DestinationIndex := IndexCheck;
			DestinationState := 0;
			EXIT;
		END_IF
	END_FOR
	IF SorterLogEnable.SORTER_DESTINATION_LU THEN
		sMessage := CONCAT('Dest ID: ', DINT_TO_STRING(DestinationID));
		sMessage := CONCAT(sMessage,' Idx: ');
		sMessage := CONCAT(sMessage, DINT_TO_STRING(DestinationIndex));
		// Write to the Error List
		ADSLOGSTR( msgCtrlMask := ADSLOG_MSGTYPE_HINT OR ADSLOG_MSGTYPE_LOG
			, msgFmtStr := 'Lookup %s'
			, strArg := sMessage);
	END_IF
END_IF

END_FUNCTION_BLOCK

// ---- POUs/Sorter_P2140.TcPOU
PROGRAM Sorter_P2140

VAR_IN_OUT
	In_ItemToInduct					: ST_Item;
	In_InductingItem				: ST_Item;
	st_tempItem						: ST_ItemTemporary;	// Temporary record used when barcode not yet received
	{attribute 'OPC.UA.DA' := '0'}
	st_Sorter						: ST_Sorter;
	{attribute 'OPC.UA.DA' := '0'}
	aDiverts						: ARRAY[Sorter.DIVERTMIN_P2140..Sorter.NUMBEROFDIVERTS_P2140] OF ST_DIVERT;
	aItems 							: ARRAY[Sorter.SORTERENCODERMIN_P2140..Sorter.SORTERENCODERMAX_P2140] OF ST_Item;
END_VAR

VAR_INPUT
	ItemsArrayMax		: UDINT;
	ItemsArrayMin		: UDINT;
	DivertArrayMax		: DINT;
	DivertArrayMin		: DINT;
END_VAR

VAR_OUTPUT
	st_DischargeItem	:	ST_Item;
END_VAR
VAR
	// Sorter Diagnostics
	aSorterDiagLog		: ST_ItemLogBuffer;
	fbSorterDiagLog		: FB_ItemLogBuffer;

	//Logging Variables
	UpdateSorterLog : FB_UpdateLog;
	
	//Induct Variables
	testEncoderCount		: UDINT;
	exitEncoderCount		: UDINT;
	lastCompareCount		: UDINT;
	updatingEncoderCount	: UDINT;

	tailendcount		: DINT := 0;
	inductindex 		: DINT;
	
	//Divert Variables
	{attribute 'OPC.UA.DA' := '0'}
	fb_DivertDecision 		: FB_DivertDecision;
	{attribute 'OPC.UA.DA' := '0'}
	fb_DivertFullMonitor  	: FB_DivertFullMonitor;
	DivertIndex				: DINT;
	Divertoffset			: INT;
	nTestItemIndex			: UDINT;
	Output2ItemIndex		: UDINT;

	// Confirm Check variables
	fb_ConfirmCheck 		: ARRAY[Sorter.DIVERTMIN_P2140..Sorter.NUMBEROFDIVERTS_P2140] OF FB_ConfirmCheck;
	st_ConfirmItem 			: ARRAY[Sorter.DIVERTMIN_P2140..Sorter.NUMBEROFDIVERTS_P2140] OF ST_Item;
	nConfirmItemIndex 		: UDINT;
	
	workingItem			: ST_Item;	// Actual item to induct

	LastItemInducted 	: STRING;
	nIndexToClear		: UDINT;	// Clear Item Array at this index
	nItemArraySize		: UDINT;

	rInductPE			: R_TRIG; 	// Capture the Rising edge of the Induct PE
	fInductPE			: F_TRIG; 	// Capture the Falling edge of the Induct PE
	sMessage			: STRING;

	st_DisplayItem		:st_Item;
	
	LogSorterDump: BOOL := FALSE;
END_VAR

// Initialize FB_ItemExtBuffer
fbSorterDiagLog(st_BufferData := aSorterDiagLog);

(*
// Test visu variables	
inductPE := SorterInductPE;
ItemsOut := Items;
ArrivalOut := ArrivalBuffer;
// End test variables
*)
(*
	Capture the Upper/Lower bound of relevant IO_OUT arrays for looping purposes
	ItemsArrayMax/Min for the sorter array slot count
*)
// Size is Max - Min + 1 to capture both extremes
nItemArraySize := ItemsArrayMax - ItemsArrayMin + 1;

FOR divertIndex := DivertArrayMin TO DivertArrayMax DO
	fb_DivertFullMonitor(Divert := aDiverts[divertIndex]);
END_FOR

(*
	Detect barcode receipt after item is already in Item array
	the tempItem is reset when the induct PE is cleared
	The tempItem is populated when the induct PE is blocked and there
	is not an associated barcode waiting to be inducted
*)
IF st_tempItem.Item.ID <> '' THEN
	// Test the IN_ItemToInduct.ID for a value
	// This record will be cleared as soon as it reaches the sorter loop
	IF In_ItemToInduct.ID <> '' THEN
		// The tempItem is overwritten with the IN_ItemToInduct after it is updated
		// But the starting encoder count is not changed so the same items can be updated
		// if the destination update is received while the item is still being inducted
		IF In_ItemToInduct.ID <> st_tempItem.Item.ID THEN 
			// Set the starting count for the testing/updating process
			// The testEncodeCount is incremented upon start, so we start -1 of the encoder count for the item
			testEncoderCount := f_CalculateIndex(Offset := -1, InitialValue:= st_tempItem.Counts, BufferSize := nItemArraySize);
			// Clear the length and start over
			In_ItemToInduct.Length := 0;
			st_tempItem.Item := In_ItemToInduct;
		END_IF 
		// Test for a change of destination after the barcode data has been received
		IF In_ItemToInduct.Destination <> st_tempItem.Item.Destination THEN 
			// Set the starting count for the testing/updating process
			// The testEncodeCount is incremented upon start, so we start -1 of the encoder count for the item
			testEncoderCount := f_CalculateIndex(Offset := -1, InitialValue:= st_tempItem.Counts, BufferSize := nItemArraySize);
			// Clear the length and start over
			In_ItemToInduct.Length := 0;
			// Copy the IN_ItemToInduct to prevent running this until something else in the record changes
			st_tempItem.Item := IN_ItemToInduct;
		END_IF
	END_IF 
END_IF


// Test for the rising edge of the induct PE
// Use this rising edge to log the IN_ItemToInduct record
rInductPE(CLK:= st_Sorter.InductPE, Q =>);

IF rInductPE.Q THEN
	IF .nSorterLogEnable.SORTER_INDUCT THEN
		sMessage := CONCAT('Item: ', In_ItemToInduct.ID);
		sMessage := CONCAT(sMessage, ' Pulses: ');
		sMessage := CONCAT(sMessage, UDINT_TO_STRING(st_Sorter.EncoderCounts));
		// Write to the Error List
		ADSLOGSTR( msgCtrlMask := ADSLOG_MSGTYPE_HINT OR ADSLOG_MSGTYPE_LOG
			, msgFmtStr := CONCAT(st_sorter.Config.Name, ' Induct Info: %s')
			, strArg := sMessage);
	END_IF
END_IF
// Test for the falling edge of the induct PE
// Use this falling edge to clear the IN_ItemToInduct record
fInductPE(CLK:= st_Sorter.InductPE, Q =>);

IF fInductPE.Q THEN
	IF .nSorterLogEnable.SORTER_INDUCT THEN
		sMessage := CONCAT('Item: ', In_ItemToInduct.ID);
		sMessage := CONCAT(sMessage,' Pulses: ');
		sMessage := CONCAT(sMEssage, UDINT_TO_STRING(st_Sorter.EncoderCounts));
		// Write to the Error List
		ADSLOGSTR( msgCtrlMask := ADSLOG_MSGTYPE_HINT OR ADSLOG_MSGTYPE_LOG
			, msgFmtStr := CONCAT(st_sorter.Config.Name, ' Cleared Induct Info: %s')
			, strArg := sMessage);
	END_IF
	// Clear the record
	In_InductingItem :=  BlankItem;
END_IF

// Process every array index between the current index and the last processed index
WHILE st_Sorter.EncoderCounts <> testEncoderCount DO

	// Capture the lastEncoderCount before changing it for comparison of last inducted items
	lastCompareCount := testEncoderCount;

	// Increment the testEncoderCount
	// The testEncoderCount variable will be used throughout the processing to ensure
	//	that all array elements are processed
	testEncoderCount := f_CalculateIndex(Offset := 1, InitialValue:= testEncoderCount, BufferSize := nItemArraySize);
	IF st_Sorter.InductPE THEN
	  	IF (In_ItemToInduct.ID <> '') THEN
			In_InductingItem := In_ItemToInduct;
			In_ItemToInduct := BlankItem;
			IF .nSorterLogEnable.SORTER_INDUCT_PE THEN
				sMessage := CONCAT('Item: ', In_InductingItem.ID);
				sMessage := CONCAT(sMessage,' Pulses: ');
				sMessage := CONCAT(sMessage, UDINT_TO_STRING(st_Sorter.EncoderCounts));
				sMessage := CONCAT(sMessage,' Dest: ');
				sMessage := CONCAT(sMessage, DINT_TO_STRING(In_InductingItem.Destination));
				sMessage := CONCAT(sMessage,' DestIdx: ');
				sMessage := CONCAT(sMessage, DINT_TO_STRING(In_InductingItem.DestinationIdx));
				// Write to the Error List
				ADSLOGSTR( msgCtrlMask := ADSLOG_MSGTYPE_HINT OR ADSLOG_MSGTYPE_LOG
					, msgFmtStr := CONCAT(st_sorter.Config.Name, ' Inducting Info: %s')
					, strArg := sMessage);
			END_IF
		END_IF
	  	IF (In_InductingItem.ID <> '') THEN
			LastItemInducted := In_InductingItem.ID;
			IF aItems[testEncoderCount].ID <> '' THEN
				IF aItems[testEncoderCount].Status >= E_StatusCode.Diverting AND aItems[testEncoderCount].Status <= E_StatusCode.Divert_UnknownError THEN
					aItems[testEncoderCount].Status := E_StatusCode.Divert_UnknownError;
				END_IF
				UpdateSorterLog(Status := aItems[testEncoderCount].Status, ItemID := aItems[testEncoderCount].UniqueID);
			END_IF
		
			// Set the Item status
			In_InductingItem.Status := E_StatusCode.In_Sorter;

			// Check for destination full on the first pass, then ignore it.
			IF In_InductingItem.Length = 0 THEN
				IF aDiverts[In_InductingItem.DestinationIdx].Full THEN
					IF st_Sorter.Config.RecircUsed THEN
						In_InductingItem.Destination := st_Sorter.Config.RecircDestination;
						In_InductingItem.DestinationIdx := st_Sorter.Config.RecircDestIdx;
						In_InductingItem.ExtStatus := E_StatusCode.Divert_Recirculated;
					ELSE
						In_InductingItem.Destination := st_Sorter.Config.DefaultDestination;
						In_InductingItem.DestinationIdx := st_Sorter.Config.DefaultDestIdx;
						In_InductingItem.ExtStatus := E_StatusCode.Divert_Full;
					END_IF
				END_IF
			END_IF
			// Clear the extend counter
			tailendcount := 0;

			// Copy the ItemToInduct to the WorkingItem that will be inducted
			workingItem := In_InductingItem;
			// Increment the Length on the ItemToInduct record, then it will be added to the array
			//  and the length will increment
			In_InductingItem.Length := In_InductingItem.Length +  1;
			// Determined by UniqueID = 0
		ELSE //If the item makes it to the sorter, but is not identified, induct the item with tempItem.Item
			LastItemInducted := 'UNKNOWN';
			UpdateSorterLog(Status := E_StatusCode.UnidentifiedItem, ItemID := st_tempItem.Item.UniqueID);

			// Process this the first time
			IF st_tempItem.Item.Length = 0 THEN
				IF nSorterLogEnable.SORTER_INDUCT_PE THEN
					sMessage := CONCAT('Temp Item: ', st_tempItem.Item.ID);
					sMessage := CONCAT(sMessage,' Pulses: ');
					sMessage := CONCAT(sMessage, UDINT_TO_STRING(st_Sorter.EncoderCounts));
					sMessage := CONCAT(sMessage,' Dest: ');
					sMessage := CONCAT(sMessage, DINT_TO_STRING(st_tempItem.Item.Destination));
					sMessage := CONCAT(sMessage,' DestIdx: ');
					sMessage := CONCAT(sMessage, DINT_TO_STRING(st_tempItem.Item.DestinationIdx));
					// Write to the Error List
					ADSLOGSTR( msgCtrlMask := ADSLOG_MSGTYPE_HINT OR ADSLOG_MSGTYPE_LOG
						, msgFmtStr := CONCAT(st_sorter.Config.Name, ' Inducting Info: %s')
						, strArg := sMessage);
				END_IF
				IF aDiverts[st_Sorter.Config.DefaultDestIdx].Full THEN
					IF st_Sorter.Config.RecircUsed THEN
						st_tempItem.Item.Destination := st_Sorter.Config.RecircDestination;
						st_tempItem.Item.DestinationIdx := st_Sorter.Config.RecircDestIdx;
						st_tempItem.Item.ExtStatus := E_StatusCode.Divert_Recirculated;
					ELSE
						st_tempItem.Item.Destination := st_Sorter.Config.DefaultDestination;
						st_tempItem.Item.DestinationIdx := st_Sorter.Config.DefaultDestIdx;
						st_tempItem.Item.ExtStatus := E_StatusCode.Divert_Full;
					END_IF
				ELSE
					st_tempItem.Item.Destination := st_Sorter.Config.DefaultDestination;
					st_tempItem.Item.DestinationIdx := st_Sorter.Config.DefaultDestIdx;
				END_IF		
			END_IF
			// Copy the tempItem.Item to the WorkingItem that will be inducted
			workingItem := st_tempItem.Item;
			// Increment the Length on the ItemToInduct record, then it will be added to the array
			//  and the length will increment
			st_tempItem.Item.Length := st_tempItem.Item.Length +  1;
		END_IF

		// Induct everything
		aItems[testEncoderCount] := workingItem;
		fbSorterDiagLog.AddItem(workingItem);
	// Follow this path when the induct photo-eye is cleared
	ELSE
		// Extend the end of the item by a set amount, or to a mimimum length
		// Test to verify that the Item index is clear, and we are still extending the length of the item
		IF aItems[lastCompareCount].ID <> '' THEN
			IF tailendcount < st_Sorter.Config.TailEndLength AND st_Sorter.Config.TailEndLength > 0 THEN
				aItems[testEncoderCount] := aItems[lastCompareCount]; 
				fbSorterDiagLog.AddItem(aItems[lastCompareCount]);
				aItems[testEncoderCount].Length := aItems[testEncoderCount].Length + 1;
				tailendcount := tailendcount + 1;
			END_IF
			IF aItems[lastCompareCount].Length < st_Sorter.Config.MinimumLength AND st_Sorter.Config.MinimumLength > 0 THEN
				aItems[testEncoderCount] := aItems[lastCompareCount]; 
				fbSorterDiagLog.AddItem(aItems[lastCompareCount]);
				aItems[testEncoderCount].Length := aItems[testEncoderCount].Length + 1;
			END_IF
		END_IF
	END_IF
END_WHILE

// Process every array index between the current index and the last processed exit index
WHILE st_Sorter.EncoderCounts <> exitEncoderCount DO

	// Increment the exitEncoderCount
	// The exitEncoderCount variable will be used throughout the processing to ensure
	//	that all array elements are processed
	exitEncoderCount := f_CalculateIndex(Offset := 1, InitialValue:= exitEncoderCount, BufferSize := nItemArraySize);
	// Process the diverts relative to the current encoder count
	FOR divertIndex := DivertArrayMin TO DivertArrayMax DO
		// Get the distance to each divert, distance is the number of pulses to actuation
		Divertoffset := aDiverts[divertIndex].Config.Distance;
		// Calculate the index of the item to test for a divert
		// Subtract the offset from the current encoder count (exitEncoderCount)
		// As the encoder count increases, the current index pointer advances
		// Subtracting looks backwards into the sorter item array to test for items at the diverts
		//	distance that should be diverted
		nTestItemIndex := F_CalculateIndex(initialvalue := exitEncoderCount
										, offset := -(Divertoffset)
										, BufferSize := (ItemsArrayMax + 1));	
		//Setup Out2Item for energizing 2nd divert output
		Output2ItemIndex := F_CalculateIndex(initialvalue := exitEncoderCount
										, offset := -(Divertoffset + UINT_TO_INT(st_Sorter.Config.Output2Offset))
										, BufferSize := (ItemsArrayMax + 1));	
		// Log Diverts
		IF aItems[nTestItemIndex].DestinationIdx = divertIndex THEN
			IF .nSorterLogEnable.SORTER_DIVERTS THEN
				sMessage := CONCAT('Item: ', aItems[nTestItemIndex].ID);
				sMessage := CONCAT(sMessage,' Index: ');
				sMessage := CONCAT(sMessage, UDINT_TO_STRING(nTestItemIndex));
				sMessage := CONCAT(sMessage,' Dest: ');
				sMessage := CONCAT(sMessage, DINT_TO_STRING(aItems[nTestItemIndex].Destination));
				sMessage := CONCAT(sMessage,' DestIdx: ');
				sMessage := CONCAT(sMessage, DINT_TO_STRING(aItems[nTestItemIndex].DestinationIdx));
				sMessage := CONCAT(sMessage,' Divert Status: ');
				sMessage := CONCAT(sMessage, DINT_TO_STRING(aDiverts[DivertIndex].Status));
				sMessage := CONCAT(sMessage,' Item Status: ');
				sMessage := CONCAT(sMessage, DINT_TO_STRING(aItems[nTestItemIndex].Status));
				// Write to the Error List
				ADSLOGSTR( msgCtrlMask := ADSLOG_MSGTYPE_HINT OR ADSLOG_MSGTYPE_LOG
					, msgFmtStr := CONCAT(st_sorter.Config.Name, ' Item at Divert Index: %s')
					, strArg := sMessage);
			END_IF
		END_IF
		fb_DivertDecision( bLog := .nDivertLogEnable.DIVERT_DECISION 
					 , Output1Item		:= aItems[nTestItemIndex]
					 , Output2Item		:= aItems[Output2ItemIndex]
					 , Divert 			:= aDiverts[DivertIndex]
					 , DivertIndex		:= DivertIndex
					 );
		// Calculate the distance to the confirm PE to test for a successful divert
		nConfirmItemIndex := F_CalculateIndex(initialvalue := exitEncoderCount
										, offset := -(Divertoffset + aDiverts[divertIndex].Config.ConfirmDist)
										, BufferSize := (ItemsArrayMax + 1));
		// Log Confirms
		IF aItems[nConfirmItemIndex].Status >= E_StatusCode.Diverting
		   AND aItems[nConfirmItemIndex].Status <= E_StatusCode.Divert_Complete
		   AND aItems[nConfirmItemIndex].UniqueID <> 0
		   AND aItems[nConfirmItemIndex].DestinationIdx = DivertIndex
		   THEN
			IF .nSorterLogEnable.SORTER_CONFIRMS THEN
				sMessage := CONCAT('Item: ', aItems[nConfirmItemIndex].ID);
				sMessage := CONCAT(sMessage,' Index: ');
				sMessage := CONCAT(sMessage, UDINT_TO_STRING(nConfirmItemIndex));
				sMessage := CONCAT(sMessage,' Dest: ');
				sMessage := CONCAT(sMessage, DINT_TO_STRING(aItems[nConfirmItemIndex].Destination));
				sMessage := CONCAT(sMessage,' DestIdx: ');
				sMessage := CONCAT(sMessage, DINT_TO_STRING(aItems[nConfirmItemIndex].DestinationIdx));
				sMessage := CONCAT(sMessage,' Divert Status: ');
				sMessage := CONCAT(sMessage, DINT_TO_STRING(aDiverts[DivertIndex].Status));
				sMessage := CONCAT(sMessage,' Item Status: ');
				sMessage := CONCAT(sMessage, DINT_TO_STRING(aItems[nTestItemIndex].Status));
				// Write to the Error List
				ADSLOGSTR( msgCtrlMask := ADSLOG_MSGTYPE_HINT OR ADSLOG_MSGTYPE_LOG
					, msgFmtStr := CONCAT(st_sorter.Config.Name, ' Item at Confirm Index: %s')
					, strArg := sMessage);
			END_IF
		END_IF
		fb_ConfirmCheck[divertIndex] ( bLog := .nDivertLogEnable.DIVERT_DECISION 
					 , ConfirmItem		:= aItems[nConfirmItemIndex]
					 , ConfirmPE 		:= aDiverts[DivertIndex].ConfirmPE
					 , DivertIndex		:= DivertIndex
					 , bIsDischarge		:= aDiverts[DivertIndex].Config.IsDischarge
					 , DetectedItem => st_ConfirmItem[DivertIndex]
					 );
	END_FOR
	
	// Capture the last item discharged by this sorter section
	IF st_ConfirmItem[DivertArrayMax].ID <> '' THEN
		st_DischargeItem := st_ConfirmItem[DivertArrayMax];
	END_IF

	// Clear the Item array ahead of the current encoder count
	nIndexToClear := f_CalculateIndex(Offset := 40, InitialValue:= exitEncoderCount, BufferSize := nItemArraySize);
	IF aItems[nIndexToClear].ID <> '' THEN
		IF .nSorterLogEnable.SORTER_DUMP THEN
			sMessage := CONCAT('Item: ', aItems[nIndexToClear].ID);
			sMessage := CONCAT(sMessage,' Index: ');
			sMessage := CONCAT(sMessage, UDINT_TO_STRING(nIndexToClear));
			sMessage := CONCAT(sMessage,' Item Status: ');
			sMessage := CONCAT(sMessage, DINT_TO_STRING(aItems[nIndexToClear].Status));
			// Write to the Error List
			ADSLOGSTR( msgCtrlMask := ADSLOG_MSGTYPE_HINT OR ADSLOG_MSGTYPE_LOG
				, msgFmtStr := CONCAT(st_sorter.Config.Name, ' Clear Ahead Dump Info: %s')
				, strArg := sMessage);
		END_IF
	END_IF
	aItems[nIndexToClear] := BlankItem;

END_WHILE

END_PROGRAM

// ---- FunctionBlocks/Item/FB_ItemLogBuffer.TcPOU
FUNCTION_BLOCK FB_ItemLogBuffer
VAR_IN_OUT
	st_BufferData	:	ST_ItemLogBuffer;	// Buffer Type	
END_VAR
VAR_INPUT
END_VAR
VAR_OUTPUT
	// Output the In and Out pointer to allow testing of the 
END_VAR
VAR
	nOutPointer		:	UDINT;				// OutPointer use to detect items in the buffer
	nBufferSizeTemp : 	UDINT;				// Calculate buffer size from Byte count
	nBufferSize : 	UDINT;					// Buffer Size in total elements
	st_Blank	:	ST_Item :=  (ID := ''
								, UniqueID := 0
								, Destination := 0
								, DestinationIdx := 0
								, Status := E_StatusCode.No_Status
								, ExtStatus := E_StatusCode.No_Status
								, DeviceID := ''
								, MessageType := E_MessageIds.NoMessage_00);
	nInit		:	UDINT;					// Used to initialize the Array on Start-up
	nItemExtSize	:	UDINT;				// Size of ST_ItemExt in Bytes
	bInitDone	: BOOL := FALSE;			// Set if Init occurred outside of FB_init
END_VAR

VAR CONSTANT
	nBITCOUNT: UINT := 32;	// Number of Bits in each Array Element
	nBYTECOUNT : UINT := 4;	// Number of Bytes in each array element
	nUDINTBYTECOUNT : UINT := 4;	// Number of Bytes in a UDINT data type
END_VAR

// This will run if FB_init did not detect a valid reference and initialize the Structure
IF nInit = 0 THEN
	// Get the Data Item In Bytes
	nBufferSizeTemp := TO_UDINT(SIZEOF(st_BufferData));
	// Reduce the byte count by the In and Out pointer byte count
	nBufferSizeTemp := nBufferSizeTemp - (nUDINTBYTECOUNT);
	// Get the size of the ST_ItemExt Data type
	nItemExtSize := TO_UDINT(SIZEOF(st_Blank));
	// Get the total number of bytes in the Array, by dividing the remaining nBufferSize by the nItemExtSize
	nBufferSize := nBufferSizeTemp/nItemExtSize;
	// Clear the Buffer on Start-up because we don't know what is and is not in process
	FOR nInit := 0 TO (nBufferSize - 1) DO
		st_BufferData.aBufferData[nInit] := st_Blank;
	END_FOR 
	// Clear the Buffer In and Out pointers
	st_BufferData.nInPointer := 0;
	nOutPointer := 0;
	// Indicate that initialization occurred outside of FB_Init
	bInitDone := TRUE;
END_IF

METHOD PUBLIC AddItem : ST_Item
VAR_INPUT
	st_ItemToAdd	:	ST_Item;
END_VAR
// Disable the warning regarding invalid Reference from a method for IO_OUT variables
{warning disable C0371}
// Test for a Valid reference
IF __ISVALIDREF(st_BufferData) THEN
	// Increment the In Pointer using the F_CaclculateIndex
	st_BufferData.nInPointer := F_CalculateIndex(Offset := 1,InitialValue := st_BufferData.nInPointer, BufferSize := nBufferSize);
	// Add the Item to the Buffer
	st_BufferData.aBufferData[st_BufferData.nInPointer] := st_ItemToAdd;
END_IF
// Restore the warning regarding invalid Reference from a method for IO_OUT variables
{warning restore C0371}
END_METHOD

PROPERTY PUBLIC BufferSize : UDINT
GET
BufferSize := nBufferSize;
END_GET
END_PROPERTY

PROPERTY PUBLIC OutPointer : UDINT
GET
OutPointer := nOutPointer;
END_GET
END_PROPERTY

METHOD PUBLIC RemoveItem : ST_Item
VAR_OUTPUT
	st_ItemToReturn	:	ST_Item;
END_VAR
// Disable the warning regarding invalid Reference from a method for IO_OUT variables
{warning disable C0371}
// Test for a Valid reference
IF __ISVALIDREF(st_BufferData) THEN
	// Increment the In Pointer using the F_CaclculateIndex
	nOutPointer := F_CalculateIndex(Offset := 1,InitialValue := nOutPointer, BufferSize := nBufferSize);
	// Add the Item to the Buffer
	st_ItemToReturn := st_BufferData.aBufferData[nOutPointer];
END_IF
// Restore the warning regarding invalid Reference from a method for IO_OUT variables
{warning restore C0371}
END_METHOD

END_FUNCTION_BLOCK

// ---- FunctionBlocks/Logging/FB_UpdateLog.TcPOU
FUNCTION_BLOCK FB_UpdateLog
VAR CONSTANT
	sizeofLog : INT := 100;
END_VAR
VAR_INPUT
	Status : E_StatusCode;
	ItemID : DINT;
END_VAR
VAR_OUTPUT
END_VAR
VAR
	StatusDescriptions :  ARRAY[0..100] OF WSTRING;
	StatusLog : ARRAY[0..sizeofLog] OF ST_LogMsg;
	GetTime : GETSYSTEMTIME;
	PLCTime : T_FILETIME;
	Time_String : STRING(24);
	LogIndex : INT;
END_VAR

(*	No_Status				:= 0,
	OK						:= 1,
	Stopped					:= 2,
	Faulted					:= 3,	
	UnknownError	 		:= 9,	*)
StatusDescriptions[E_StatusCode.No_Status] 				:= "No_Status - This is the default status";
StatusDescriptions[E_StatusCode.OK] 						:= "OK - The system is OK";
StatusDescriptions[E_StatusCode.Stopped] 					:= "Stopped - The system is stopped";
StatusDescriptions[E_StatusCode.Faulted]					:= "Faulted - The system is faulted";
StatusDescriptions[E_StatusCode.UnknownError] 				:= "UnknownError - There is an unknown error with the system";

(*	NotInSorter				:= 20,	
	UpdateRequested			:= 21,
	QueryNeeded				:= 22,
	UpdateNeeded 			:= 23,
	UpdateReceived 			:= 24,
	ReqNotReceived			:= 25,
	ItemNotUpdated			:= 26,
	UnidentifiedItem		:= 27,
	ItemNotFound			:= 28,
	Sorter_UnknownError 	:= 29,
	Assign_Accepted			:= 30,
	Assign_Full				:= 31,
	Assign_NotFound			:= 32,
	Assign_NotInducted		:= 33, *)
StatusDescriptions[E_StatusCode.NotInSorter] 				:= "NotInSorter - This item is Not in the Sorter";
StatusDescriptions[E_StatusCode.UpdateRequested] 			:= "UpdateRequested - This item has requested an update";
StatusDescriptions[E_StatusCode.QueryNeeded] 				:= "QueryNeeded - This item requires an query";
StatusDescriptions[E_StatusCode.UpdateNeeded] 				:= "UpdateNeeded - This item requires an update";
StatusDescriptions[E_StatusCode.UpdateReceived] 			:= "UpdateReceived - This item received an update";
StatusDescriptions[E_StatusCode.ReqNotReceived]			:= "ReqNotReceived - This item never received an update. Make the buffer bigger?";
StatusDescriptions[E_StatusCode.ItemNotUpdated] 			:= "ItemNotUpdated - Item left sorter before receiving information update";
StatusDescriptions[E_StatusCode.UnidentifiedItem] 			:= "UnidentifiedItem - There might be an item in the sorter that is not identified";
StatusDescriptions[E_StatusCode.ItemNotFound] 				:= "ItenNotFound - Item not found on the Sorter";
StatusDescriptions[E_StatusCode.Sorter_UnknownError] 		:= "Sorter_UnknownError - Something happened to an item while in the sorter";
StatusDescriptions[E_StatusCode.Assign_Accepted] 			:= "Assign_Accepted - Destination Assignment Accepted";
StatusDescriptions[E_StatusCode.Assign_Full] 				:= "Assign_Full - Destination Assignment Unavailable, full, offline, or faulted";
StatusDescriptions[E_StatusCode.Assign_NotFound] 			:= "Assign_NotFound - Assignment Failed, Item not Found";
StatusDescriptions[E_StatusCode.Assign_NotInducted] 		:= "Assign_NotInducted - Item not inducted before new item detected";

(*	In_Sorter 				:= 41,
	Diverting 				:= 42,
	Divert_Success 			:= 43,
	Divert_Full				:= 44,
	Divert_Offline			:= 45,
	Divert_Missed 			:= 46,
	Divert_Failed 			:= 47,
	Divert_NotInducted		:= 48,
	Divert_UnknownError 	:= 49, *)
StatusDescriptions[E_StatusCode.In_Sorter] 				:= "In_Sorter - This item is in the sorter";
StatusDescriptions[E_StatusCode.Diverting] 				:= "Diverting - This item is diverting";
StatusDescriptions[E_StatusCode.Divert_Success] 			:= "Divert_Success - This item successfully diverted";
StatusDescriptions[E_StatusCode.Divert_Full] 				:= "Divert_Full - Assigned Divert Lane Full";
StatusDescriptions[E_StatusCode.Divert_Offline] 			:= "Divert_Offline - Assigned Divert Lane Offline";
StatusDescriptions[E_StatusCode.Divert_Missed] 			:= "Divert_Missed - This item missed its divert";
StatusDescriptions[E_StatusCode.Divert_Recirculated] 			:= "Divert_Recirculated - This item was Recirculated";
StatusDescriptions[E_StatusCode.Divert_NotInducted] 		:= "Divert_NotInducted - Item not inducted before new item detected";
StatusDescriptions[E_StatusCode.Divert_UnknownError] 		:= "Divert_UnknownError - Something happened to this item while diverting";

(*	In_Transfer 			:= 61,
	Transferring 			:= 62,
	Tranfer_Success	 		:= 63,
	Transfer_Missed 		:= 64,
	Transfer_Failed 		:= 65,	
	Transfer_UnknownError 	:= 69 *)
StatusDescriptions[E_StatusCode.In_Transfer] 				:= "In_Transfer - This item is in the transfer area";
StatusDescriptions[E_StatusCode.Transferring] 				:= "Transferring - This item is transferring";
StatusDescriptions[E_StatusCode.Tranfer_Success] 			:= "Tranfer_Success - This item successfully transferred";
StatusDescriptions[E_StatusCode.Transfer_Missed] 			:= "Transfer_Missed - This item missed its transfer";
StatusDescriptions[E_StatusCode.Transfer_Failed] 			:= "Transfer_Failed - This item failed to transfer";
StatusDescriptions[E_StatusCode.Transfer_UnknownError] 	:= "Transfer_UnknownError - Something happened to this item while transferring";


FOR LogIndex := sizeofLog TO 1 BY -1 DO
		StatusLog[Logindex] := StatusLog[LogIndex-1];
END_FOR

GetTime(timeLoDW=>PLCTime.dwLowDateTime, timeHiDW=>PLCTime.dwHighDateTime);

StatusLog[0].DateandTime := SystemTIME_TO_STRING(FILETIME_TO_SYSTEMTIME(PLCTime));
StatusLog[0].ItemID := ItemID;
StatusLog[0].Status := Status;
StatusLog[0].StatusDescription := StatusDescriptions[Status];

END_FUNCTION_BLOCK

// ---- FunctionBlocks/Divert/Functions/FB_DivertDecision.TcPOU
FUNCTION_BLOCK FB_DivertDecision
VAR_IN_OUT
	Output1Item 		: ST_Item;
	Output2Item			: ST_Item;
	Divert 				: ST_Divert;
END_VAR

VAR_INPUT
	DivertIndex 		: DINT;
	bLog				: BOOL;
END_VAR

VAR
	DivertController	: FB_DivertControl;
	Output1Activate 	: BOOL := 0;
	Output2Activate 	: BOOL := 0;	
	UpdateLog 			: FB_UpdateLog;
	LastDest 			: DINT;	
	aDivertLog			: ST_ItemLogBuffer;
	fbDivertLog			: FB_ItemLogBuffer;
	ItemToLog			: ST_Item;
	sMessage			: STRING;
END_VAR

fbDivertLog(st_BufferData := aDivertLog);

//Divert this item if this divert is this item's intended destination
IF DivertIndex = Output1Item.DestinationIdx THEN
	// Check this only once, then set the Status accordingly
	IF Divert.Status = E_StatusCode.Divert_Idle THEN
		IF Divert.Full THEN
			Divert.Status := E_StatusCode.Divert_Full;
		else
			Divert.Status := E_StatusCode.Diverting;
		END_IF
		IF bLog THEN
			sMessage := CONCAT('Item: ', Output1Item.ID);
			sMessage := CONCAT(sMessage,' Dest: ');
			sMessage := CONCAT(sMessage, DINT_TO_STRING(Output1Item.Destination));
			sMessage := CONCAT(sMessage,' Status: ');
			sMessage := CONCAT(sMessage, DINT_TO_STRING(Divert.Status));
			// Write to the Error List
			ADSLOGSTR( msgCtrlMask := ADSLOG_MSGTYPE_HINT OR ADSLOG_MSGTYPE_LOG
				, msgFmtStr := CONCAT(Divert.Config.ID, ' Divert Initiated: %s')
				, strArg := sMessage);
		END_IF
	END_IF;
	IF Divert.Status = E_StatusCode.Diverting THEN
		Output1Activate := 1;
		Divert.Item := Output1Item;
		//Energize Output2 after SorterCode.CFG_Output2Offset has passed 
		IF DivertIndex = Output2Item.DestinationIdx THEN
			Output2Activate := 1;
		END_IF
		DivertController( Output1Activate	:= Output1Activate
				, Output2Activate	:= Output2Activate
				, Output1Item		:= Output1Item
				, Output2Item		:= Output2Item
				, Divert			:= Divert
				);		
	ELSIF Divert.Status = E_StatusCode.Divert_Full THEN
		Output1Item.ExtStatus := E_StatusCode.Divert_Full;
	END_IF				
//	Output1Item.Status := Divert.Status; 
	ItemToLog := Output1Item;
	ItemToLog.Length := DivertIndex;
	fbDivertLog.AddItem(ItemToLog);
ELSE
	//Turn off output if dest does not equal divert index
	Output1Activate := 0;
	//Keep Output2 energized for SorterCode.CFG_Output2Offset distance
	IF DivertIndex <> Output2Item.DestinationIdx THEN
		// Set and Idle status for the divert
		Divert.Status := E_StatusCode.Divert_Idle;
		Output2Activate := 0;
	ELSE
		Output2Activate := 1;	
	END_IF	

	DivertController( Output1Activate	:= Output1Activate
				, Output2Activate	:= Output2Activate
				, Output1Item		:= Output1Item
				, Output2Item		:= Output2Item
				, Divert			:= Divert
				);
END_IF

END_FUNCTION_BLOCK

// ---- FunctionBlocks/Divert/Functions/FB_DivertControl.TcPOU
FUNCTION_BLOCK FB_DivertControl
VAR_IN_OUT
	Divert			: ST_Divert;
	Output1Item 	: ST_Item ;
	Output2Item 	: ST_Item ;
END_VAR

VAR_INPUT
	Output1Activate	: BOOL;	
	Output2Activate	: BOOL;	 
END_VAR

VAR
	Test : BOOL;
END_VAR

(*
	This function block exists to 
	energize the physical outputs
	of a diverter. 
*)

IF Output1Activate THEN
	Divert.Output1 := 1;	
	Test := 1;
	IF Output1Item.Status < E_StatusCode.Diverting THEN
		Output1Item.Status := E_StatusCode.Diverting;
		Output1Item.DeviceID := Divert.Config.EquipID;
	END_IF
ELSE
	Divert.Output1 := 0;
END_IF
	
IF Output2Activate THEN
	Divert.Output2 := 1;	
	IF Output2Item.Status < E_StatusCode.Diverting THEN
		Output2Item.Status := E_StatusCode.Diverting;
		Output2Item.DeviceID := Divert.Config.EquipID;
	END_IF
ELSE
	Divert.Output2 := 0;				
END_IF

END_FUNCTION_BLOCK

// ---- FunctionBlocks/Divert/Functions/FB_DivertFullMonitor.TcPOU
FUNCTION_BLOCK FB_DivertFullMonitor

VAR_IN_OUT
	Divert 			: ST_Divert;
END_VAR

VAR
	LastFullTime	: REAL;
	nFullTime : UINT;
	Cfg_FullTime: TIME := T#2S;
END_VAR

// Calculate and set the merge clear timer
IF LastFullTime <> Divert.Config.FullTime THEN
	LastFullTime := Divert.Config.FullTime;
	nFullTime := REAL_TO_UINT(LastFullTime * 1000); 
	Cfg_FullTime := UINT_TO_TIME(nFullTime);
END_IF

// Set the Full time, according to the Full-Time
Divert.FullTimer(PT := Cfg_FullTime);

// Test for Full
Divert.FullTimer(IN := Divert.FullPE);

IF Divert.FullTimer.Q THEN
	IF NOT Divert.Full THEN
		IF nDivertLogEnable.LANEFULL THEN
			// Write to the Error List
			ADSLOGSTR( msgCtrlMask := ADSLOG_MSGTYPE_HINT OR ADSLOG_MSGTYPE_LOG
				, msgFmtStr := CONCAT(STR1 := Divert.Config.ID, STR2 := ' Full: %s')
				, strArg := CONCAT (STR1 := ' Item: ', STR2 := Divert.Item.ID));
		END_IF
	END_IF
	Divert.Full := TRUE;
ELSE
	IF Divert.Full THEN
		IF nDivertLogEnable.LANEFULL THEN
			// Write to the Error List
			ADSLOGSTR( msgCtrlMask := ADSLOG_MSGTYPE_HINT OR ADSLOG_MSGTYPE_LOG
				, msgFmtStr := CONCAT(STR1 := Divert.Config.ID, STR2 := ' Not Full: %s')
				, strArg := CONCAT (STR1 := ' Item: ', STR2 := Divert.Item.ID));
		END_IF
	END_IF
	Divert.Full := FALSE;
END_IF

END_FUNCTION_BLOCK

// ---- FunctionBlocks/Divert/Functions/FB_ConfirmCheck.TcPOU
(*
	Each confirm location needs its own instance of this FunctionBlock in order to allow the LastDest to corretly detect sorted items
	
	No faults are set in this routine, it just checks for items at confirm PE's when they are expected/not expected

	DetecetedItem is set when the item has blocked and then cleared the confirm PE
*)
FUNCTION_BLOCK FB_ConfirmCheck
VAR_IN_OUT
	ConfirmItem 		: ST_Item;
END_VAR

VAR_INPUT
	ConfirmPE			: BOOL;
	DivertIndex 		: DINT;
	bIsDischarge		: BOOL;
	bLog				: BOOL;
END_VAR

VAR_OUTPUT
	DetectedItem		: ST_Item;
END_VAR

VAR
	UpdateLog 			: FB_UpdateLog;
	LastDest 			: DINT;	
	aDivertLog			: ST_ItemLogBuffer;
	fbDivertLog			: FB_ItemLogBuffer;
	ItemToLog			: ST_Item;
	sMessage			: STRING;
	BlankItem					: ST_Item := (ID := '', UniqueID := 0
													, Destination := 0
													, DestinationIdx := 0
													, Status := E_StatusCode.No_Status
													, ExtStatus := E_StatusCode.No_Status
													, DeviceID := ''
													, MessageType := E_MessageIds.NoMessage_00);

END_VAR

// Clear the Detected Item each iteration to ensure that it only has a item assigned after the confirm PE has been cleared
DetectedItem := BlankItem;

// Check Confirm item. If it was marked diverting
// Only check if the item is valid
IF ConfirmPE THEN 
	IF (ConfirmItem.Status >= E_StatusCode.Diverting AND ConfirmItem.Status <= E_StatusCode.Divert_Complete)
	   AND ConfirmItem.UniqueID <> 0 THEN
		// Set the Status to Divert_Detected, because we see the item
		//	ProcesBuffer will propogate that status
		ConfirmItem.Status := E_StatusCode.Divert_Detected;
		// The first time around, create a log item
		IF LastDest = 0 THEN
			UpdateLog(Status := ConfirmItem.Status, ItemID := ConfirmItem.UniqueID);
			ItemToLog := ConfirmItem;
			ItemToLog.Length := DivertIndex;
			fbDivertLog.AddItem(ItemToLog);
		END_IF
//		DetectedItem := ConfirmItem;
		// Capture the Current item destination before exiting the function block to test against the next run
		LastDest := ConfirmItem.Destination;
	END_IF
ELSE
	// If we had a valid item, because we have a LastDest, set the Divert_Success to true under certain conditions
	//	And write to the log
	IF LastDest > 0 THEN
		IF ConfirmItem.Status = E_StatusCode.Divert_Detected THEN
			ConfirmItem.Status := E_StatusCode.Divert_Success;
			DetectedItem := ConfirmItem;
			// Set a divert missed status if this is a discharge and the destination does not match the index
			IF bIsDischarge THEN
				IF DetectedItem.Destination <> DivertIndex AND ConfirmItem.ExtStatus = 0 THEN
					ConfirmItem.ExtStatus := E_StatusCode.Divert_Missed;
				END_IF
			END_IF
			// Log when the item clears the confirm PE
			UpdateLog(Status := DetectedItem.Status, ItemID := DetectedItem.UniqueID);
			ItemToLog := DetectedItem;
			ItemToLog.Length := DivertIndex;
			fbDivertLog.AddItem(ItemToLog);
		END_IF
		LastDest := 0;
	END_IF
END_IF

END_FUNCTION_BLOCK

// ---- POUs/ProcessBuffers_P2150.TcPOU
PROGRAM ProcessBuffers_P2150
VAR_IN_OUT
	st_NextToInduct					: ST_ItemTemporary;
	st_UpdateItem					: ST_ItemTemporary;
	st_TempInductItem				: ST_ItemTemporary;
	{attribute 'OPC.UA.DA' := '0'}
	st_Sorter						: ST_Sorter;
	{attribute 'OPC.UA.DA' := '0'}
	aDiverts						: ARRAY[Sorter.DIVERTMIN_P2150..Sorter.NUMBEROFDIVERTS_P2150] OF ST_DIVERT;
	aItems 							: ARRAY[Sorter.SORTERENCODERMIN_P2150..Sorter.SORTERENCODERMAX_P2150] OF ST_Item;
END_VAR

VAR_INPUT
	DivertToCommission				: DINT;
	ItemsArrayMax 			: UDINT;
	ItemsArrayMin 			: UDINT;
END_VAR

VAR_OUTPUT
	DefaultDestIdx					: DINT;
	RecircDestIdx					: DINT;
END_VAR

VAR
	fb_ArrivalBuffer				: FB_ItemBuffer;
	st_ArrivalItem 					: ST_Item;		// Arrival Item (Bar code read) from System PLC (BarCodeReaders.pou)

	// Item to replace in the sorter buffer
	st_ReplaceItem					: st_Item;

	fb_TransportBuffer				: FB_ItemBuffer;

	fb_UpdateBuffer 				: FB_ItemBuffer;

	st_ToUpdate						: ST_ItemTemporary;	// Item to Update on the Sorter, or waiting to be added to the sorter

	ItemsArraySize			: UDINT;

	TransportItemInSorter	: ST_Item;	// Temporary Processing Item
	TransportItemFound		: ST_Item;	// Item to Update Found
	TransportSorterIndex	: UDINT;

	ExitSorterIndex			: UDINT;
	ExitItemInSorter		: ST_Item;
	ExitItemFound			: ST_ItemTemporary;
	ExitInDivert			: BOOL;
	ExitDiverting			: BOOL;
	ExitSuccess				: BOOL;
	ExitDetected			: BOOL;
	ExitComplete			: BOOL;

	UpdateIndexCounter		: DINT;

	bTest : BOOL;
	sMessage	:	STRING;
	
	st_DisplayItem		:st_Item;
	LogSorterDump		:BOOL := FALSE;
	fb_FindDestination		: FB_FindDestination;
	fb_DefaultDestination	: FB_FindDestination;
	fb_RecircDestination	: FB_FindDestination;
	// Created to allow the aDiverts to be used in the FB_FindDestination Function Block
	{attribute 'OPC.UA.DA' := '0'}
	aTempDiverts			: ARRAY[Sorter.DIVERTMIN_P2150..Sorter.NUMBEROFDIVERTS_P2150] OF ST_DIVERT;
	
	nItemBufferLogEnable	:	UDINT;
	nSorterLogEnable		:	UDINT;
	nDivertLogEnable		:	UDINT;
	nSortBufferLogEnable	:	UDINT;
END_VAR

nItemBufferLogEnable := GVL_Logging.nItemBufferLogEnable OR GVL_Logging.nItemBufferLogEnableP2150;
nSorterLogEnable := GVL_Logging.nSorterLogEnable OR GVL_Logging.nSorterLogEnableP2150;
nDivertLogEnable := GVL_Logging.nDivertLogEnable OR GVL_Logging.nDivertLogEnableP2150;
nSortBufferLogEnable := GVL_Logging.nSortBufferLogEnable OR GVL_Logging.nSortBufferLogEnableP2150;

aTempDiverts := aDiverts;
// Initialize the Transport and Update buffers
// Set Master for FB's that control the buffer
fb_ArrivalBuffer.Master := FALSE;
fb_TransportBuffer.Master := FALSE;
fb_UpdateBuffer.Master := TRUE;

// Turn ON/OFF Logging of all activity in/out
fb_ArrivalBuffer.LogEntries := .nItemBufferLogEnable.ARRIVALS;
fb_TransportBuffer.LogEntries := .nItemBufferLogEnable.TRANSPORT;
fb_UpdateBuffer.LogEntries := .nItemBufferLogEnable.UPDATE;

// Provide names for the buffers
fb_ArrivalBuffer.Name := '2150 SRT ARRIVAL';
fb_TransportBuffer.Name := '2150 SRT TRANSPORT';
fb_UpdateBuffer.Name := '2150 SRT UPDATE';

// Initialize the FB_ItemExtBuffer Instances
fb_ArrivalBuffer(st_BufferData := st_SorterArrivalBuffer_P2150
						, st_BufferFdbkIn := st_ArrivalFdbkOut_P2150
						, st_BufferFdbkOut => st_ArrivalFdbkIn_P2150);
fb_TransportBuffer(st_BufferData := st_SorterTransportBuffer_P2150
						, st_BufferFdbkIn := st_TransportFdbkOut_P2150
						, st_BufferFdbkOut => st_TransportFdbkIn_P2150);
fb_UpdateBuffer(st_BufferData := st_SorterUpdateBuffer
						, st_BufferFdbkIn := st_UpdateFdbkIn
						, st_BufferFdbkOut => st_UpdateFdbkOut);

IF GVL_IO.INIT THEN
	fb_ArrivalBuffer.Clear();
	fb_TransportBuffer.Clear();
	fb_UpdateBuffer.Clear();
END_IF
						
(*
	Set the Upper/Lower bound of relevant arrays for looping purposes
	ItemsArrayMax/Min for the sorter array slot count
*)
// Size is Max - Min + 1 to capture both extremes
ItemsArraySize := ItemsArrayMax - ItemsArrayMin + 1;

(*
 	Check for a value disagreement in the Arrival Buffer In and Out pointers to
  	determine if there is an update for an item.
	When an Item arrives, the System PLC adds it to the shared buffer and increments
	the InPointer
*)
IF st_SorterArrivalBuffer_P2150.nInPointer <> fb_ArrivalBuffer.OutPointer THEN
	fb_ArrivalBuffer.RemoveItem(st_ItemToReturn => st_ArrivalItem);
END_IF

// Input Item read at bar code reader from System PLC to sorter
IF st_ArrivalItem.ID <> '' THEN
	IF .nSortBufferLogEnable.BUFFER_ARRIVAL THEN
		sMessage := CONCAT(' Item: ', st_ArrivalItem.ID);
		sMessage := CONCAT(sMessage,' Pulses: ');
		sMessage := CONCAT(sMessage, UDINT_TO_STRING(st_Sorter.EncoderCounts));
		// Write to the Error List
		ADSLOGSTR( msgCtrlMask := ADSLOG_MSGTYPE_HINT OR ADSLOG_MSGTYPE_LOG
			, msgFmtStr := 'Arrival Processed: %s'
			, strArg := sMessage);
	END_IF
	// Indicate that this item did not get added to the sorter and add to the exit buffer
	//  Both as a TransportUpdate and TransportComplete message type 
	IF st_NextToInduct.Item.ID <> '' THEN
		IF .nSortBufferLogEnable.BUFFER_MISSINDUCT THEN
			sMessage := CONCAT(' Item: ', st_NextToInduct.Item.ID);
			// Write to the Error List
			ADSLOGSTR( msgCtrlMask := ADSLOG_MSGTYPE_HINT OR ADSLOG_MSGTYPE_LOG
				, msgFmtStr := 'Item Removed - Not Inducted: %s'
				, strArg := sMessage);
		END_IF
		// Transport Response
		st_NextToInduct.Item.Status := E_StatusCode.Assign_NotInducted;
		st_NextToInduct.Item.DeviceID := st_Sorter.Config.EquipID;
		st_NextToInduct.Item.MessageType := E_MessageIds.TransportResponse_25;
		fb_UpdateBuffer.AddItem(st_ItemToAdd := st_NextToInduct.Item);

		// Transport Complete
		st_NextToInduct.Item.Status := E_StatusCode.Divert_NotInducted;
		st_NextToInduct.Item.MessageType := E_MessageIds.TransportComplete_26;
		fb_UpdateBuffer.AddItem(st_ItemToAdd := st_NextToInduct.Item);
	END_IF
	// Copy Last BCR item to Item to Induct
	st_NextToInduct.Item :=  st_ArrivalItem;
	// Add the Sorter EquipID to the NextToInduct
	st_NextToInduct.Item.DeviceID := st_Sorter.Config.EquipID;
	// Set the Default Destination
	st_NextToInduct.Item.Destination := st_Sorter.Config.DefaultDestination;
	st_NextToInduct.Item.DestinationIdx := st_Sorter.Config.DefaultDestIdx;
	// Capture an encoder value that when the encoder count exceeds this value, NextToInduct item will be cleared
	st_NextToInduct.Counts := st_Sorter.EncoderCounts;
	// Clear the Last recieved item
	st_ArrivalItem := BlankItem;
	// Prepare to replace the Temporarily assigned item with this item
	IF st_TempInductItem.Item.ID <> '' THEN
		// Capture the Counts and Length from the temporary item
		st_NextToInduct.Counts := st_TempInductItem.Counts;
		st_NextToInduct.Item.Length := st_TempInductItem.Item.Length;
		//Identify the Item to replace in the sorter array
		st_ReplaceItem := st_TempInductItem.Item;
		st_TempInductItem.Counts := 0;
		st_TempInductItem.Item := BlankItem;
		IF .nSortBufferLogEnable.BUFFER_TEMPINDUCT THEN
			ADSLOGSTR( msgCtrlMask := ADSLOG_MSGTYPE_HINT OR ADSLOG_MSGTYPE_LOG
				, msgFmtStr := 'Temp ID Replaced : %s'
				, strArg := st_ReplaceItem.ID); 
		END_IF
	END_IF
END_IF

(*
 	Check for a value disagreement in the SorterTransportBuffer In and Out pointers to
  	determine if there is an update for an item.
	When an update arrived, the System PLC adds it to the shared buffer and increments
	the InPointer
*)
IF st_SorterTransportBuffer_P2150.nInPointer <> fb_TransportBuffer.OutPointer THEN
	fb_TransportBuffer.RemoveItem(st_ItemToReturn => st_ToUpdate.Item);
	// Lookup the index for the chosen destination
	fb_FindDestination(RoundRobin := st_Sorter.Config.RoundRobin
					, SorterLogEnable := .nSorterLogEnable
					, aDiverts := aTempDiverts
					, DestinationID := st_ToUpdate.Item.Destination
					, DestinationIndex => st_ToUpdate.Item.DestinationIdx);
	IF .nSortBufferLogEnable.BUFFER_DESTINDEX THEN
		sMessage := CONCAT(' Item: ', st_ToUpdate.Item.ID);
		sMessage := CONCAT(sMessage,' Destination: ');
		sMessage := CONCAT(sMessage, DINT_TO_STRING(st_ToUpdate.Item.Destination));
		sMessage := CONCAT(sMessage,' Index: ');
		sMessage := CONCAT(sMessage, DINT_TO_STRING(st_ToUpdate.Item.DestinationIdx));
		// Write to the Error List
		ADSLOGSTR( msgCtrlMask := ADSLOG_MSGTYPE_HINT OR ADSLOG_MSGTYPE_LOG
			, msgFmtStr := 'Divert Index of Destination: %s'
			, strArg := sMessage);
	END_IF
END_IF

// Get the Default Destination Index
fb_DefaultDestination(RoundRobin := st_Sorter.Config.RoundRobin
				, aDiverts := aTempDiverts
				, DestinationID := st_Sorter.Config.DefaultDestination
				, DestinationIndex => DefaultDestIdx);

// Get the Recirculation Destination Index
fb_RecircDestination(RoundRobin := st_Sorter.Config.RoundRobin
				, aDiverts := aTempDiverts
				, DestinationID := st_Sorter.Config.RecircDestination
				, DestinationIndex => RecircDestIdx);

// Test the Item to Update against the Item to Induct and update if they match:
//	Update the NextItemToInduct with the updated data, then clear the Item to Update
IF st_ToUpdate.Item.ID <> '' THEN
	IF st_ToUpdate.Item.ID = st_NextToInduct.Item.ID THEN
		// Indicate that the transport command was received and a response was sent
		st_NextToInduct.Item.MessageType := E_MessageIds.TransportResponse_25;
		// Test the assigned lane for availability
		IF aDiverts[st_ToUpdate.Item.DestinationIdx].Full
		   OR aDiverts[st_ToUpdate.Item.DestinationIdx].Faulted THEN
			// Prepare a message to indicate that the item cannot be assigned
			st_ToUpdate.Item.Status := E_StatusCode.Assign_Full;
			st_ToUpdate.Item.DeviceID := st_Sorter.Config.EquipID;
			st_ToUpdate.Item.MessageType := E_MessageIds.TransportResponse_25;
			fb_UpdateBuffer.AddItem(st_ItemToAdd := st_ToUpdate.Item);
			st_NextToInduct.Item.ExtStatus := E_StatusCode.Divert_Full;
		ELSE
			st_NextToInduct.Item.DeviceID := st_Sorter.Config.EquipID;
			st_NextToInduct.Item.Status := E_StatusCode.Assign_Accepted;
			// Update the Destination
			st_NextToInduct.Item.Destination := st_ToUpdate.Item.Destination;
			st_NextToInduct.Item.DestinationIdx := st_ToUpdate.Item.DestinationIdx;
			fb_UpdateBuffer.AddItem(st_ItemToAdd := st_NextToInduct.Item);
		END_IF
		// If commissioning, ignore any other direction
		IF DivertToCommission > 0 THEN
			st_NextToInduct.Item.Destination := DivertToCommission;
		END_IF
		// Log the update
		IF .nSortBufferLogEnable.BUFFER_INDUCT THEN
			sMessage := CONCAT(' Item: ', st_ToUpdate.Item.ID);
			sMessage := CONCAT(sMessage,' Pulses: ');
			sMessage := CONCAT(sMessage, UDINT_TO_STRING(st_Sorter.EncoderCounts));
			sMessage := CONCAT(sMessage,' Status: ');
			sMessage := CONCAT(sMessage, UDINT_TO_STRING(st_ToUpdate.Item.Status));
			sMessage := CONCAT(sMessage,' Ext Status: ');
			sMessage := CONCAT(sMessage, UDINT_TO_STRING(st_ToUpdate.Item.ExtStatus));
			// Write to the Error List
			ADSLOGSTR( msgCtrlMask := ADSLOG_MSGTYPE_HINT OR ADSLOG_MSGTYPE_LOG
				, msgFmtStr := 'Found Before Induct: %s'
				, strArg := sMessage);
		END_IF
		// We updated the item we were inducting, clear the Item to update
		st_ToUpdate.Item := BlankItem;
	END_IF
END_IF

// Clear the Update Item Found record each pass
TransportItemFound := BlankItem;

// Clear the last detected Exit item
ExitItemFound.Item := BlankItem;

// Reset the Detection booleans
ExitInDivert := FALSE;
ExitDiverting := FALSE;
ExitDetected := FALSE;
ExitSuccess := FALSE;
ExitComplete := FALSE;

// Loop through the entire array, it should be appropriately sized for the length of the sorter section
FOR UpdateIndexCounter := UDINT_TO_DINT(ItemsArrayMin) TO UDINT_TO_DINT(ItemsArrayMax) DO //Loop through everything in the sorter	

	// For Transport commands, start from the current encoder count and work forwards, just like the exit
	TransportSorterIndex := F_CalculateIndex(Offset := (UpdateIndexCounter)
											, InitialValue := st_Sorter.EncoderCounts
											, BufferSize := ItemsArraySize);

	// This is the item in the sorter array that we will be procesing this pass, testing for a Transport update message
	TransportItemInSorter := aItems[UDINT_TO_DINT(TransportSorterIndex)];

	// Test for a replace item
	// ReplaceItem is the temporary item
	// NextToInduct is the item to replace the temporary with
	IF st_ReplaceItem.ID <> '' THEN
		IF st_ReplaceItem.ID = TransportItemInSorter.ID THEN
			IF .nSortBufferLogEnable.BUFFER_REPLACEINDUCT THEN
				sMessage := CONCAT(' Item: ', st_ReplaceItem.ID);
				sMessage := CONCAT(sMessage,' New Item: ');
				sMessage := CONCAT(sMessage, st_NextToInduct.Item.ID);
				sMessage := CONCAT(sMessage,' Index: ');
				sMessage := CONCAT(sMessage, UDINT_TO_STRING(TransportSorterIndex));
				sMessage := CONCAT(sMessage,' Orig Dest: ');
				sMessage := CONCAT(sMessage, DINT_TO_STRING(TransportItemInSorter.Destination));
				sMessage := CONCAT(sMessage,' New Dest: ');
				sMessage := CONCAT(sMEssage, DINT_TO_STRING(st_ReplaceItem.Destination));
				sMessage := CONCAT(sMessage,' Orig Idx: ');
				sMessage := CONCAT(sMessage, DINT_TO_STRING(TransportItemInSorter.DestinationIdx));
				sMessage := CONCAT(sMessage,' New Idx: ');
				sMessage := CONCAT(sMEssage, DINT_TO_STRING(st_ReplaceItem.DestinationIdx));
				// Write to the Error List
				ADSLOGSTR( msgCtrlMask := ADSLOG_MSGTYPE_HINT OR ADSLOG_MSGTYPE_LOG
					, msgFmtStr := 'Item ID Replaced After Induct: %s'
					, strArg := sMessage);
			END_IF
			TransportItemInSorter.ID := st_NextToInduct.Item.ID;
			TransportItemInSorter.Destination := st_NextToInduct.Item.Destination;
			TransportItemInSorter.DestinationIdx := st_NextToInduct.Item.DestinationIdx;
			TransportItemInSorter.DeviceID := st_NextToInduct.Item.DeviceID;
			TransportItemInSorter.MessageType := st_NextToInduct.Item.MessageType;
			TransportItemInSorter.Status := st_NextToInduct.Item.Status;
			TransportItemInSorter.UniqueID := st_NextToInduct.Item.UniqueID;
			TransportItemInSorter.CapturedInMetrics := st_NextToInduct.Item.CapturedInMetrics;
		END_IF
	END_IF
	// Test for an Item Update
	IF st_ToUpdate.Item.ID <> '' THEN
		// Test the sorter item against the update item
		IF st_ToUpdate.Item.ID = TransportItemInSorter.ID THEN
			IF .nSortBufferLogEnable.BUFFER_UPDATEINDUCT THEN
				sMessage := CONCAT(' Item: ', st_ToUpdate.Item.ID);
				sMessage := CONCAT(sMessage,' Index: ');
				sMessage := CONCAT(sMessage, UDINT_TO_STRING(TransportSorterIndex));
				// Write to the Error List
				ADSLOGSTR( msgCtrlMask := ADSLOG_MSGTYPE_HINT OR ADSLOG_MSGTYPE_LOG
					, msgFmtStr := 'Found After Induct: %s'
					, strArg := sMessage);
			END_IF
			// Copy the found item record, 
			TransportItemFound := TransportItemInSorter;
			// Test the destined divert for availability
			IF aDiverts[st_ToUpdate.Item.DestinationIdx].Full OR aDiverts[st_ToUpdate.Item.DestinationIdx].Faulted THEN
				// Prepare a message to indicate that the item cannot be assigned
				TransportItemFound.Status := E_StatusCode.Assign_Full;
				TransportItemFound.ExtStatus := E_StatusCode.Divert_Full;
				TransportItemFound.MessageType := E_MessageIds.TransportResponse_25;
				TransportItemFound.Destination := st_Sorter.Config.DefaultDestination;
				TransportItemFound.DestinationIdx := st_Sorter.Config.DefaultDestIdx;
			// Test for an already diverting item and assign an ExtStatus of LateAssignment
			ELSIF TransportItemInSorter.Status >= E_StatusCode.Diverting THEN
				TransportItemFound.ExtStatus := E_StatusCode.Divert_LateAssignment;
				TransportItemFound.MessageType := E_MessageIds.TransportResponse_25;
			ELSE
				//  Change the destination, which should be the only item in the update
				TransportItemFound.Destination := st_ToUpdate.Item.Destination;
				TransportItemFound.DestinationIdx := st_ToUpdate.Item.DestinationIdx;
				// This message indicates we could assign the Item
				TransportItemFound.Status := E_StatusCode.Assign_Accepted;
				TransportItemFound.MessageType := E_MessageIds.TransportResponse_25;
			END_IF
			TransportItemFound.DeviceID := st_Sorter.Config.EquipID;
			// Add the item to the update buffer
			fb_UpdateBuffer.AddItem(TransportItemFound);
			// Clear the ToUpdate Item
			st_ToUpdate.Item := BlankItem;
		END_IF
	END_IF
	
	IF TransportItemFound.ID <> '' THEN
		// Test the sorter item against the update item
		IF TransportItemFound.ID = TransportItemInSorter.ID THEN
			// Only update if it is different
			IF TransportItemFound.Destination <> TransportItemInSorter.Destination THEN
				IF .nSortBufferLogEnable.BUFFER_UPDATEDEST THEN
					sMessage := CONCAT(' Item: ', TransportItemInSorter.ID);
					sMessage := CONCAT(sMessage,' Index: ');
					sMessage := CONCAT(sMessage, UDINT_TO_STRING(TransportSorterIndex));
					sMessage := CONCAT(sMessage,' Orig Dest: ');
					sMessage := CONCAT(sMessage, DINT_TO_STRING(TransportItemInSorter.Destination));
					sMessage := CONCAT(sMessage,' Orig Idx: ');
					sMessage := CONCAT(sMessage, DINT_TO_STRING(TransportItemInSorter.DestinationIdx));
					sMessage := CONCAT(sMessage,' Orig DeviceID ');
					sMessage := CONCAT(sMessage, TransportItemInSorter.DeviceID);
					// Write to the Error List
					ADSLOGSTR( msgCtrlMask := ADSLOG_MSGTYPE_HINT OR ADSLOG_MSGTYPE_LOG
						, msgFmtStr := 'Dest Updated After Induct: %s'
						, strArg := sMessage);
				END_IF
				// Update the Destination. If the destination is unavailable, it has been already been set to the default
				TransportItemInSorter.Destination := TransportItemFound.Destination;
				TransportItemInSorter.DestinationIdx := TransportItemFound.DestinationIdx;
				TransportItemInSorter.DeviceID := TransportItemFound.DeviceID;
				TransportItemInSorter.MessageType := TransportItemFound.MessageType;
				TransportItemInSorter.Status := TransportItemFound.Status;
				TransportItemInSorter.ExtStatus := TransportItemFound.ExtStatus;
	
				IF .nSortBufferLogEnable.BUFFER_UPDATEDEST THEN
					sMessage := CONCAT(' Item: ', TransportItemInSorter.ID);
					sMessage := CONCAT(sMessage,' Index: ');
					sMessage := CONCAT(sMessage, UDINT_TO_STRING(TransportSorterIndex));
					sMessage := CONCAT(sMessage,' New Dest: ');
					sMessage := CONCAT(sMessage, DINT_TO_STRING(TransportItemInSorter.Destination));
					sMessage := CONCAT(sMessage,' New Idx: ');
					sMessage := CONCAT(sMessage, DINT_TO_STRING(TransportItemInSorter.DestinationIdx));
					sMessage := CONCAT(sMessage,' New DeviceID ');
					sMessage := CONCAT(sMessage, TransportItemInSorter.DeviceID);
					// Write to the Error List
					ADSLOGSTR( msgCtrlMask := ADSLOG_MSGTYPE_HINT OR ADSLOG_MSGTYPE_LOG
						, msgFmtStr := 'Dest Updated After Induct: %s'
						, strArg := sMessage);
				END_IF
			END_IF
			// Make sure that the destination update makes it to the item being inducted into the sorter
			IF st_UpdateItem.Item.ID <> '' THEN
				IF st_UpdateItem.Item.ID = TransportItemFound.ID THEN
					IF st_UpdateItem.Item.Destination <> TransportItemFound.Destination THEN
						IF .nSortBufferLogEnable.BUFFER_UPDATEDEST THEN
							// Log the original destination
							sMessage := CONCAT(' Item: ', st_UpdateItem.Item.ID);
							sMessage := CONCAT(sMessage, ' Pulses: ');
							sMessage := CONCAT(sMessage, UDINT_TO_STRING(st_Sorter.EncoderCounts));
							sMessage := CONCAT(sMessage,' Orig Dest: ');
							sMessage := CONCAT(sMessage, DINT_TO_STRING(st_UpdateItem.Item.Destination));
							sMessage := CONCAT(sMessage,' Orig Idx: ');
							sMessage := CONCAT(sMessage, DINT_TO_STRING(st_UpdateItem.Item.DestinationIdx));
							// Write to the Error List
							ADSLOGSTR( msgCtrlMask := ADSLOG_MSGTYPE_HINT OR ADSLOG_MSGTYPE_LOG
								, msgFmtStr := 'Induct Dest Changed: %s'
								, strArg := sMessage);
						END_IF
						// Update the Destination and Index
						st_UpdateItem.Item.Destination := TransportItemFound.Destination;
						st_UpdateItem.Item.DestinationIdx := TransportItemFound.DestinationIdx;
						// Log the new destination
						IF .nSortBufferLogEnable.BUFFER_UPDATEDEST THEN
							sMessage := CONCAT(' Item: ', st_UpdateItem.Item.ID);
							sMessage := CONCAT(sMessage, ' Pulses: ');
							sMessage := CONCAT(sMessage, UDINT_TO_STRING(st_Sorter.EncoderCounts));
							sMessage := CONCAT(sMessage,' New Dest: ');
							sMessage := CONCAT(sMessage, DINT_TO_STRING(st_UpdateItem.Item.Destination));
							sMessage := CONCAT(sMessage,' New Idx: ');
							sMessage := CONCAT(sMessage, DINT_TO_STRING(st_UpdateItem.Item.DestinationIdx));
							// Write to the Error List
							ADSLOGSTR( msgCtrlMask := ADSLOG_MSGTYPE_HINT OR ADSLOG_MSGTYPE_LOG
								, msgFmtStr := 'Induct Dest Changed: %s'
								, strArg := sMessage);
						END_IF
					END_IF
				END_IF
			ELSE
				IF .nSortBufferLogEnable.BUFFER_UPDATEDEST THEN
					sMessage := CONCAT(' Item: ', TransportItemInSorter.ID);
					sMessage := CONCAT(sMessage,' Index: ');
					sMessage := CONCAT(sMessage, UDINT_TO_STRING(TransportSorterIndex));
					sMessage := CONCAT(sMessage,' Orig Dest: ');
					sMessage := CONCAT(sMessage, DINT_TO_STRING(TransportItemInSorter.Destination));
					sMessage := CONCAT(sMessage,' Orig Idx: ');
					sMessage := CONCAT(sMessage, DINT_TO_STRING(TransportItemInSorter.DestinationIdx));
					// Write to the Error List
					ADSLOGSTR( msgCtrlMask := ADSLOG_MSGTYPE_HINT OR ADSLOG_MSGTYPE_LOG
						, msgFmtStr := 'Dest Received After Induct: %s'
						, strArg := sMessage);
				END_IF	
			END_IF
		END_IF
	END_IF

	// Put the updated record back into the array
	aItems[TransportSorterIndex] := TransportItemInSorter;
	
//==================================================
// 	Done procesing Transport information
//
//	Begin processing Update/Exit information
//==================================================
	
	// For exits, start from the current encoder count and work forward
	ExitSorterIndex := F_CalculateIndex(Offset := UpdateIndexCounter
										, InitialValue := st_Sorter.EncoderCounts
										, BufferSize := ItemsArraySize);

	// Identify the Item we are testing
	ExitItemInSorter := aItems[ExitSorterIndex];

